	STATE_HV_ON:				BOOL;			(*Haute tension en marche*)
	STATE_HV:					BOOL;			(*Demande de mise en marche de la Haute Tension en cours*)
	STATE_SRC_ON:				BOOL;			(*Source en marche*)
	STATE_SRC:					BOOL;			(*Demande de mise en marche de la source en cours*)
	STATE_NOK:					BOOL;			(*Alimentation en défaut*)
	STATE_I_Fil:				REAL;			(*Mesure Courant filament (A)*)
	STATE_V_HV:					REAL;			(*Mesure de la tension (kV)*)
	STATE_I_EMISS:				REAL;			(*Mesure du courant d'émission (mA)*)
	STATE_COURANT:				REAL;			(* Courant appliqué en % *)
	STATE_READY:				BOOL;
END_VAR

VAR
END_VAR

HV.IdParent := MNEMO;
SRC.IdParent := MNEMO;
HV.IdXML := '16';
HV.TagXML := 1;
SRC.IdXML := '16';
SRC.TagXML := 2;
HV.MNEMO := 	CONCAT(MNEMO,'_HV');
SRC.MNEMO :=	CONCAT(MNEMO,'_SRC');

(*Défaut*)
HV.DEF_Off.IdXML				:=	'3';
HV.DEF_Off.TagXML				:=	3;
HV.DEF_On.IdXML				:=	'3';
HV.DEF_On.TagXML				:=	1;
HV.DEF_Off_Auto.IdXml			:=	'3';
HV.DEF_Off_Auto.TagXml			:=	10;
HV.DEF_On_imposs.IdXml		:=	'3';
HV.DEF_On_imposs.TagXml		:=	5;
HV.DEF_Off_imposs.IdXml		:=	'3';
HV.DEF_Off_imposs.TagXml		:=	8;

SRC.DEF_Off.IdXML				:=	'3';
SRC.DEF_Off.TagXML			:=	3;
SRC.DEF_On.IdXML				:=	'3';
SRC.DEF_On.TagXML			:=	1;
SRC.DEF_Off_Auto.IdXml			:=	'3';
SRC.DEF_Off_Auto.TagXml		:=	10;
SRC.DEF_On_imposs.IdXml		:=	'3';
SRC.DEF_On_imposs.TagXml		:=	5;
SRC.DEF_Off_imposs.IdXml		:=	'3';
SRC.DEF_Off_imposs.TagXml		:=	8;


HV(
	RESET:= RESET,
	MANUAL:= MANUAL,
	IN_ON:= NOT IN_HV_ON,
	CO_On:= CO_HV,
	EN_On_INT:=DOOR AND WATER AND VAC,
	EN_Off_INT:= TRUE,
	CONF_Type_Actuator:= 0,
	CONF_EN_On:= 0,
	CONF_DI_Off:= FALSE,
	CONF_DI_On:= TRUE,
	CONF_No_Safety_Auto:= FALSE,
	CONF_Tim_Valid_On:= T#2s,
	CONF_Tim_Valid_Off:= T#50ms,
	OUT_On=>OUT_HV,
	STATE_On=> STATE_HV_ON );
	
HV.DEF_Off.DELAY := T#10s;
HV.DEF_On.DELAY := T#10s;

STATE_HV := HV.OUT_On;

SRC(
	RESET:= RESET,
	MANUAL:= MANUAL,
	CO_On:=CO_SRC,
	IN_ON:= NOT IN_SRC_ON,
	EN_On_INT:=DOOR AND WATER  AND VAC AND (I_CR_OK OR (STATE_COURANT= 0)) AND STATE_HV_ON,
	EN_Off_INT:= TRUE,
	CONF_Type_Actuator:= 0,
	CONF_EN_On:= 0,
	CONF_DI_Off:= FALSE,
	CONF_DI_On:= TRUE,
	CONF_No_Safety_Auto:=FALSE ,
	CONF_Tim_Valid_On:= T#2s,
	CONF_Tim_Valid_Off:= T#50ms,
	OUT_On=>OUT_SRC,
	STATE_On=>STATE_SRC_ON );
	
SRC.DEF_Off.DELAY := T#10s;
SRC.DEF_On.DELAY := T#10s;

STATE_SRC := SRC.OUT_On;

AI_UHV(
	CONF_Max:= 10.0,
	CONF_Min:= 0.0,
	CONF_Bipolar:=FALSE,
	CONF_Range:= 1,
	INPUT:= IN_UHVQ ,
	Value=> STATE_V_HV );

AI_IEM(
	CONF_Max:= 1000,
	CONF_Min:= 0.0,
	CONF_Bipolar:=FALSE,
	CONF_Range:= 1,
	INPUT:= IN_IEMQ,
	Value=> STATE_I_EMISS );

AI_FIL(
	CONF_Max:= 100,
	CONF_Min:= 0.0,
	CONF_Bipolar:=FALSE ,
	CONF_Range:= 1,
	INPUT:= IN_FILQ ,
	Value=> STATE_I_Fil );

(*Gestion de la sortie analogique de courant d'emission*)
IF NOT STATE_SRC_ON OR RESET THEN
	AO_QIEM.Value := 0.0;
ELSIF MANUAL THEN
	AO_QIEM.Value := PRM_COURANT;
ELSE
	AO_QIEM.Value := I_COURANT;
END_IF;
STATE_COURANT:= AO_QIEM.Value;

AO_QIEM(
	CONF_Max:=100,  (*%*)
	CONF_Min:= 0,
	CONF_Bipolar:=FALSE ,
	CONF_Range:=1 ,
	OUTPUT=> OUT_QIEM );

(*Gestion de la sortie analogique haute tension*)
IF RESET THEN
	AO_QUHV.Value := 0.0;
ELSIF MANUAL THEN
	AO_QUHV.Value := PRM_TENSION;
ELSE
	AO_QUHV.Value := I_TENSION;
END_IF;

AO_QUHV(
	CONF_Max:=10,
	CONF_Min:= 0,
	CONF_Bipolar:=FALSE ,
	CONF_Range:=1 ,
	OUTPUT=> OUT_QUHV );

(*Gestion des interlock*)
OUT_ITLCK_VAC := DOOR AND VAC;
OUT_ITLCK_HVAC := DOOR AND VAC;
OUT_ITLCK_WAT := WATER;


STATE_NOK:= HV.STATE_Nok OR SRC.STATE_Nok;
STATE_READY:= WATER AND DOOR AND VAC AND I_CR_OK;

END_FUNCTION_BLOCK

// ---- POUs/FONCTION DE BASE/ANALOG_INPUT.TcPOU
FUNCTION_BLOCK ANALOG_INPUT
(* Fonction standard AC de mise à l'échelle *)

(****************historique des versions*****************************)

(* Version 1-0 - HG - VERSION INIITIALE*)

(*************************************************************************)
VAR_INPUT  PERSISTENT
	CONF_Max:	 			REAL;				(* ~ (OPC : 1 : available for OPC-clients) *)			(*valeur min*)
	CONF_Min: 				REAL:=0.0;			(* ~ (OPC : 1 : available for OPC-clients) *)			(*valeur max*)
	CONF_Bipolar:			BOOL:= FALSE;													(*option conversion en bipolaire (+/- 10V par ex) ou non (0-10V)*)
	CONF_Range:				REAL:=1;														(*Facteur de conversion par ex 0.5 pour une entrée ana 5V = pleine echelle*)
END_VAR

VAR_INPUT
 	INPUT:				 	INT;					(* ~ (OPC : 1 : available for OPC-clients) *)			(*entrée analogique*)
END_VAR

VAR_OUTPUT
	Value:					REAL;				(* ~ (OPC : 1 : available for OPC-clients) *)			(*value analogique convertie*)
END_VAR

IF CONF_Range = 0.0 THEN
	Value	:=	0;
	RETURN;
END_IF
IF CONF_Bipolar THEN
	Value	:=	(((INT_TO_REAL(INPUT) -32768.0)  * (CONF_Max-CONF_Min) / 65535.0 )  + CONF_Min) / CONF_Range;
ELSE
	Value	:=	((INT_TO_REAL(INPUT)   * (CONF_Max-CONF_Min) / 32767.0 )  + CONF_Min) / CONF_Range;
END_IF;

END_FUNCTION_BLOCK

// ---- POUs/FONCTION DE BASE/ANALOG_OUTPUT.TcPOU
FUNCTION_BLOCK ANALOG_OUTPUT
(* Fonction standard AC de mise à l'échelle *)

(****************historique des versions*****************************)

(* Version 1-0 - SP - VERSION INIITIALE*)

(*************************************************************************)
VAR_INPUT  PERSISTENT
	CONF_Max:	 			REAL;														(*valeur min*)
	CONF_Min: 				REAL:=0.0;													(*valeur max*)
	CONF_Bipolar:			BOOL:= FALSE;												(*option conversion en bipolaire (+/- 10V par ex) ou non (0-10V)*)
	CONF_Range:				REAL:=1;													(*Facteur de conversion par ex 0.5 pour une entrée ana 5V = pleine echelle*)
END_VAR

VAR_INPUT
 	Value:					REAL;				(* ~ (OPC : 1 : available for OPC-clients) *)		(*entrée analogique*)
END_VAR

VAR_OUTPUT
	OUTPUT:					INT ;				(* ~ (OPC : 1 : available for OPC-clients) *)		(*value analogique convertie*)
END_VAR

IF (CONF_Max-CONF_Min) = 0 THEN
	OUTPUT := 0;
	RETURN;
END_IF
IF CONF_Bipolar THEN
	OUTPUT := REAL_TO_INT((((Value - CONF_Min)*65536.0 / (CONF_Max-CONF_Min))+ 32767.0) * CONF_range);
ELSE
	OUTPUT := REAL_TO_INT(((Value - CONF_Min) * 32767.0 / (CONF_Max - CONF_Min)) * CONF_Range);
END_IF;

END_FUNCTION_BLOCK

// ---- POUs/Composant/EVAP/BLOCK_SOURCE_JOULE.TcPOU
FUNCTION_BLOCK BLOCK_SOURCE_JOULE
VAR_INPUT
	DOOR:						BOOL;		(*porte fermée*)
	VAC:						BOOL;		(*sécurité vide*)
	WATER:						BOOL;		(*refroidissement source ok*)
	MANUAL:					BOOL;		(*demande mode manuel*)
	I_CR_OK:					BOOL;		(*Positionnement creuset ok*)
	RESET:						BOOL;		(*reset*)

	AI_UEJ:						ANALOG_INPUT;
	AI_IEJ:						ANALOG_INPUT;

	IN_IEJQ			AT%I*:		INT;			(* Entrée analogique courant*)
	IN_UEJQ			AT%I*:		INT;			(* Entrée analogique tension*)

	EJ:							BLOCK_ACTUATOR2;		(*Source Effet Joule*)

	I_POWER:					REAL;		(*consigne de puissance appliquée en mode automatique*)
	PRM_POWER:				REAL;		(*Consigne de puissance appliquée en mode manuel*)
	CO_SRC:					BOOL;		(*Commande externe de marche de la source en automatique*)

END_VAR

VAR_INPUT PERSISTENT
	(*Entité*)
	IsComponent:		BOOL;			(*entité : composant*)
	IdXML:			STRING;			(*nom entité : identifiant pour recherche dans dico*)
	TagXML:			UINT;			(*nom entité : identifiant pour recherche dans dico*)
	IdParent:			STRING;			(*MNEMO de l'appelant*)
	MNEMO:			STRING;			(*MNEMO de l'entité*)
END_VAR

VAR_OUTPUT
	OUT_MEJ			AT%Q*:		BOOL;		(*Marche Effet joule*)

	AO_QEJ:				ANALOG_OUTPUT;		(*Sortie analogique consigne effet joule*)
	OUT_QEJ			AT%Q*:		INT;			(*Consigne effet joule*)

	STATE_UEJ:			REAL;			
	STATE_IEJ:			REAL;			
	
	
	STATE_EJ_ON:		BOOL;			(*Etat effet joule en marche*)

	STATE_POWER:		REAL;			(*Puissance appliquée en %*)

	STATE_NOK:			BOOL;			(*Alimentation en défaut*)
	STATE_READY:		BOOL;
END_VAR
VAR
END_VAR

EJ.IdParent := MNEMO;
EJ.IdXML := '16';
EJ.TagXML := 11;
EJ.MNEMO := 	CONCAT(MNEMO,'_EJ');

(*Défaut*)
EJ.DEF_Off_Auto.IdXml			:=	'3';
EJ.DEF_Off_Auto.TagXml		:=	10;
EJ.DEF_On_imposs.IdXml		:=	'3';
EJ.DEF_On_imposs.TagXml	:=	5;
EJ.DEF_Off_imposs.IdXml		:=	'3';
EJ.DEF_Off_imposs.TagXml	:=	8;


EJ(
	RESET:= RESET,
	MANUAL:= MANUAL,
	CO_On:=CO_SRC ,
	EN_On_INT:=DOOR AND WATER AND VAC AND (I_CR_OK OR (STATE_POWER = 0)),
	EN_Off_INT:= TRUE,
	CONF_No_Safety_Auto:=FALSE ,
	CONF_EN_On:= ,
	CONF_Tim_Valid_On:= T#5s,
	CONF_Tim_Valid_Off:= T#50ms,
	OUT_On=>,
	STATE_On=> ,
	STATE_Nok=> );

(*Demande marche Effet Joule*)
OUT_MEJ:= EJ.OUT_On;
STATE_EJ_ON:= OUT_MEJ;


(*Gestion de la sortie analogique*)
IF NOT STATE_EJ_ON OR RESET THEN
	AO_QEJ.Value := 0.0;
ELSIF MANUAL THEN
	AO_QEJ.Value := PRM_POWER;
ELSE
	AO_QEJ.Value := I_POWER;
END_IF;

AO_QEJ(
	CONF_Max:=100 ,	(*%*)
	CONF_Min:= 0,
	CONF_Bipolar:=FALSE ,
	CONF_Range:=1 );
OUT_QEJ:= AO_QEJ.OUTPUT;

STATE_POWER:= AO_QEJ.Value;

(*Retour Source en défaut*)
STATE_NOK:= EJ.STATE_Nok;
STATE_READY:= WATER AND DOOR AND VAC AND I_CR_OK;

(*Gestion de la sortie analogique source effet joule *)

AI_UEJ(
	CONF_Max:= 30.0,
	CONF_Min:= 0.0,
	CONF_Bipolar:=FALSE,
	CONF_Range:= 1,
	INPUT:= IN_UEJQ ,
	Value=> STATE_UEJ );

AI_IEJ(
	CONF_Max:= 500.0,
	CONF_Min:= 0.0,
	CONF_Bipolar:=FALSE,
	CONF_Range:= 1,
	INPUT:= IN_IEJQ ,
	Value=> STATE_IEJ );

END_FUNCTION_BLOCK

// ---- POUs/Composant/EVAP/BLOCK_TELEMARK_CHEETAH_SWEEP.TcPOU
FUNCTION_BLOCK BLOCK_TELEMARK_CHEETAH_SWEEP

(* Gestion d'un controleur de balayage telemark Digital Sweep 8 motifs*)

(****************historique des versions*****************************)

(* Version 1-0 - LDS - 01/09/26 - VERSION INIITIALE EVA900 n°1 - 5236 *)


(*************************************************************************)

VAR_INPUT
	MANUAL:					BOOL;		(*Mode de pilotage manuel *)
	RESET:					BOOL;		(*Condition de réinitialisation de la fonction *)
	DOOR:					BOOL;		(*Porte fermée*)
	
	I_SW_RUN:				BOOL;		(*Balayage en marche*)
	I_SW_RDY:				BOOL;		(*Balayage prêt*)
	
	PRM_NbBal:				USINT:=1;	(*Commande de position*)
	
	CO_Remote:				BOOL;		(*Demande d'activation du mode remote en automatique*)
	CO_Balayage:			BOOL;		(*Demande d'activation du balayage*)
END_VAR

VAR
	TIMER_Valid_On:			TON;
	TIMER_Valid_Off:		TOF;
	M_Remote:				BOOL;	(* Ordre de changement commande remote *)
	RCP_M_Remote:			BOOL;	(* Bit de reception de l'ordre de remote du module de balayage*)
	VAR_Remote:				BOOL;	(* Variable intermédiaire commande remote du module de balayage*)
	
	M_balayage:				BOOL;	(* Ordre de balayage en manuel*)
	RCP_M_Balayage:			BOOL;	(* Bit de reception de l'ordre de balayage du module de balayage*)
	VAR_Balayage:			BOOL;	(* Variable intermédiaire commande balayage du module de balayage*)
END_VAR

VAR_OUTPUT
	OUT_SWB1:			BOOL;		(*sélection du motif*)
	OUT_SWB2:			BOOL;		(*sélection du motif*)
	OUT_SWB3:			BOOL;		(*sélection du motif*)
	OUT_SWB4:			BOOL;		(*sélection du motif*)
	OUT_SWP_ON:			BOOL;		(*SWEEP ON/OFF*)
	OUT_RMT:			BOOL;		(*Remote*)
	STATE_NbBal:		USINT;
	STATE_BAL:			STRING;
	STATE_REM:			BOOL;		(*Module de balayage en mode Remote*)
	STATE_LOC:			BOOL;		(*Module de balayage en mode Local*)
	STATE_ON:			BOOL;		(*Module de balayage en marche*)
	STATE_OFF:			BOOL;		(*Module de balayage à l'arrêt*)
	STATE_RDY:			BOOL;		(*Module de balayage à prêt*)
	AUTOR_Remote_IHM:			BOOL;		(*indique que le changement mode remote est autorisé en mode manuel depuis l'IHM*)
	AUTOR_Remote_PLC:			BOOL;		(*indique que le changement more remote est autorisé en mode automatique depuis l'automate*)
	AUTOR_BALAYAGE_IHM:			BOOL;		(*indique que le changement mode remote est autorisé en mode manuel depuis l'IHM*)
	AUTOR_BALAYAGE_PLC:			BOOL;		(*indique que le changement more remote est autorisé en mode automatique depuis l'automate*)
END_VAR


VAR_INPUT PERSISTENT

	PRM_BAL: 		ARRAY[0..8] OF STRING;		(*nom du programme de balayage*)

	(*Entité*)
	IsComponent:	BOOL;			(*entité : composant*)
	IdXML:			STRING;			(*nom entité : identifiant pour recherche dans dico*)
	TagXML:			UINT;			(*nom entité : identifiant pour recherche dans dico*)
	IdParent:		STRING;			(*MNEMO de l'appelant*)
	MNEMO:			STRING;			(*MNEMO de l'entité*)
END_VAR

(* Gestion des ordres en mode manuel *)
RCP_M_Remote			:=	M_Remote;
RCP_M_Balayage			:=	M_Balayage;

(*affectation des bits d'état*)
STATE_REM			:=	OUT_RMT;
STATE_LOC			:=	NOT OUT_RMT;
STATE_OFF			:=	NOT I_SW_RUN;
STATE_RDY			:=	I_SW_RDY;

(*indicateur  STATE_ON*)

TIMER_Valid_On.IN	:=	I_SW_RUN;
TIMER_Valid_On(PT:=T#500ms);
TIMER_Valid_Off.IN	:=	I_SW_RUN;
TIMER_Valid_Off(PT:=T#200ms);
STATE_ON			:=	Timer_Valid_On.Q AND TIMER_Valid_Off.Q;

(*gestion des bits d'autorisation en mode manuel*)
AUTOR_Remote_IHM		:=	NOT RESET AND MANUAL;
AUTOR_Remote_PLC		:=	NOT RESET AND NOT MANUAL;
AUTOR_Balayage_IHM		:=	NOT RESET AND MANUAL;
AUTOR_Balayage_PLC		:=	NOT RESET AND NOT MANUAL;

(*Selection du mode de balayage*)
CASE PRM_NbBal OF
		8:
			OUT_SWB1 := FALSE;
			OUT_SWB2 := FALSE;
			OUT_SWB3 := FALSE;
			OUT_SWB4 := TRUE;
		7:
			OUT_SWB1 := TRUE;
			OUT_SWB2 := TRUE;
			OUT_SWB3 := TRUE;
			OUT_SWB4 := FALSE;
		6:
			OUT_SWB1 := FALSE;
			OUT_SWB2 := TRUE;
			OUT_SWB3 := TRUE;
			OUT_SWB4 := FALSE;
		5:
			OUT_SWB1 := TRUE;
			OUT_SWB2 := FALSE;
			OUT_SWB3 := TRUE;
			OUT_SWB4 := FALSE;
		4:
			OUT_SWB1 := FALSE;
			OUT_SWB2 := FALSE;
			OUT_SWB3 := TRUE;
			OUT_SWB4 := FALSE;
		3:
			OUT_SWB1 := TRUE;
			OUT_SWB2 := TRUE;
			OUT_SWB3 := FALSE;
			OUT_SWB4 := FALSE;
		2:
			OUT_SWB1 := FALSE;
			OUT_SWB2 := TRUE;
			OUT_SWB3 := FALSE;
			OUT_SWB4 := FALSE;
		1:
			OUT_SWB1 := TRUE;
			OUT_SWB2 := FALSE;
			OUT_SWB3 := FALSE;
			OUT_SWB4 := FALSE;
END_CASE
STATE_NbBal := PRM_NbBal;
IF STATE_NbBal > 0 THEN
	STATE_BAL:= PRM_BAL[STATE_NbBal];
ELSE
	STATE_BAL:= '';
END_IF

(*gestion SWP ON*)
IF	(CO_balayage AND AUTOR_BALAYAGE_PLC)
		 OR 	(RCP_M_Balayage AND NOT VAR_BALAYAGE AND AUTOR_BALAYAGE_IHM) THEN
			VAR_BALAYAGE 		:= 	TRUE;
ELSIF (NOT Co_balayage AND NOT RESET AND NOT MANUAL)
		OR 	(RCP_M_Balayage AND VAR_BALAYAGE AND AUTOR_BALAYAGE_IHM)
		OR 	RESET THEN
			VAR_BALAYAGE		:=	FALSE;
END_IF;
OUT_SWP_ON	:=	VAR_BALAYAGE;


(*gestion remote*)
IF	(CO_Remote AND AUTOR_Remote_PLC)
		 OR 	(RCP_M_Remote AND NOT VAR_Remote AND AUTOR_Remote_IHM) THEN
			VAR_Remote 		:= 	TRUE;
ELSIF (NOT CO_Remote AND NOT RESET AND NOT MANUAL)
		OR 	(RCP_M_Remote AND VAR_Remote AND AUTOR_Remote_IHM)
		OR 	RESET THEN
			VAR_Remote		:=	FALSE;
END_IF;
OUT_RMT	:=	VAR_Remote;

(* Reset des ordres*)
IF M_Remote	AND RCP_M_Remote THEN
	M_Remote			:=	FALSE;
END_IF

(* Reset des ordres*)
IF M_Balayage AND RCP_M_Balayage THEN
	M_Balayage		:=	FALSE;
END_IF

END_FUNCTION_BLOCK

// ---- POUs/Composant/EVAP/BLOCK_IND_CR_396_TELEMARK.TcPOU
FUNCTION_BLOCK BLOCK_IND_CR_396_TELEMARK

(* Pour utilisation d'un indexeur de creuset telemark 396/398 à 6 creusets max *)

(****************historique des versions*****************************)

(* Version 0 - 21/03/19 - GV - Affaire: 11385 - Block de base : BLOCK_IND_CR_379_TELEMARK *)

(*************************************************************************)

VAR_INPUT

	MANUAL:					BOOL;		(*Mode de pilotage manuel *)
	RESET:					BOOL;		(*Condition de réiinitialisation de la fonction *)

	CO_Change:				BOOL;		(*Demande de changement de creuset en automatique*)
	CO_Remote:				BOOL;
	I_FIL_ON:				BOOL;
	PRM_NCR:				USINT:=1;	(*Commande de position*)

	IN_POWER:				REAL;		(*Puissance appliquée au creuset*)

	IN_POS1:				BOOL;		(*position de l'indexeur*)
	IN_POS2:				BOOL;
	IN_POS3:				BOOL;
	IN_POS4:				BOOL;		(*position de l'indexeur*)
	IN_POS5:				BOOL;
	IN_POS6:				BOOL;
	IN_POS_OK:				BOOL;

	DEF_POSITIONNEMENT:	PRCDEF;	(*Défaut de positionnement*)
END_VAR

VAR
	VAR_Cpt_Temps:				ARRAY[0..8] OF BLOCK_CPT_TEMPS;		(*Compteur de fonctionnement pour chaque creuset*)
	VAR_Cpt_Puissance:			ARRAY[0..8] OF BLOCK_CPT_INTEG;		(*Compteur pour chaque creuset*)
	VAR_Cpt_Epaisseur:			ARRAY[0..8] OF BLOCK_CPT_INTEG;		(*Compteur d'épaisseur pour chaque creuset*)
	I:							USINT;									(*Variable d'itération*)

	M_Change:					BOOL;	(* Ordre de changement de creuset en manuel *)
	RCP_M_Change:				BOOL;	(* Bit de reception de l'ordre de Marche/Arrêt du module de balayage *)
	VAR_Change:					BOOL;	(* Variable intermédiaire de marche du module de balayage*)
	M_Remote: 					BOOL;
	RCP_M_Remote:				BOOL;
	VAR_Remote:					BOOL;
	
	TIMER_Valid_Pos_Creuset:		TON;	(*Attentede validation du positionnement du creuset*)
	FM_CO_remote:  				R_trig;
	FM_CO_Change:				r_trig;
	VAR_Mem_CO_remote:BOOL;
	VAR_Mem_CO_change:bool;
END_VAR

VAR_OUTPUT
	AUTOR_Change_IHM:			BOOL;		(*indique que le changement de creuset est autorisée en mode manuel depuis l'IHM*)
	AUTOR_Change_PLC:			BOOL;		(*indique que le changement de creuset est autorisée en mode automatique depuis l'automate*)
	AUTOR_Remote_IHM:			BOOL;		
	AUTOR_Remote_PLC:			BOOL;
	
	OUT_SEL1:					BOOL;		(*sélection  des creusets*)
	OUT_SEL2:					BOOL;
	OUT_SEL3:					BOOL;
	OUT_SEL4:					BOOL;		(*sélection  des creusets *)
	OUT_SEL5:					BOOL;
	OUT_SEL6:					BOOL;
	OUT_RMT:					BOOL;		(*force remote*)
	STATE_ROT:					BOOL;		(*Creuset en rotation*)
	STATE_NOK:					BOOL;		(*Positionnement nok*)
	STATE_POS_OK:				BOOL;		(*Positionnement ok*)
	STATE_POS:					USINT;
	STATE_MAT:					STRING;
	STATE_REM:					BOOL;		(*Remote OK*)
END_VAR

VAR_INPUT PERSISTENT
	CONF_NCR:		USINT;	(*Nombre de creuset disponible*)

	PRM_MAT: 		ARRAY[0..8] OF STRING;		(*nom de la matière associée au creuset*)

	(*Entité*)
	IsComponent:		BOOL;			(*entité : composant*)
	IdXML:			STRING;			(*nom entité : identifiant pour recherche dans dico*)
	TagXML:			UINT;			(*nom entité : identifiant pour recherche dans dico*)
	IdParent:			STRING;			(*MNEMO de l'appelant*)
	MNEMO:			STRING;			(*MNEMO de l'entité*)
END_VAR

(*Défaut*)
DEF_POSITIONNEMENT.IdXml			:=	'14';
DEF_POSITIONNEMENT.TagXml		:=	2;


(* Gestion des ordres en mode manuel *)
	RCP_M_Change			:=	M_Change;
	RCP_M_Remote			:=  M_remote;


	
(*gestion des bits d'autorisation en mode manuel*)
	AUTOR_Change_IHM		:=	NOT RESET AND NOT Var_Change AND NOT I_FIL_ON AND MANUAL;
	AUTOR_Change_PLC		:=	NOT RESET AND NOT I_FIL_ON AND NOT MANUAL;
	AUTOR_Remote_IHM		:=	NOT RESET AND MANUAL;
	AUTOR_Remote_PLC		:=	NOT RESET AND NOT MANUAL;	

(*gestion des variables intermédiare*)

(*Changement Creuset*)
	IF	(CO_change AND AUTOR_Change_PLC AND NOT var_change)								/////////
			 OR 	( RCP_M_Change AND AUTOR_Change_IHM) THEN
				Var_Change 		:= 	TRUE;
	ELSIF (VAR_Change AND STATE_POS_OK) THEN
				Var_Change		:=	FALSE;
	END_IF;
	
(*Remote*)	
IF (CO_remote AND AUTOR_Remote_PLC AND NOT var_remote) 									/////////
	OR (RCP_M_remote AND NOT var_remote AND AUTOR_Remote_IHM) THEN
		VAR_remote:=TRUE;
ELSIF (NOT CO_remote AND NOT reset AND NOT manual ) 
		OR (RCP_M_Remote AND VAR_Remote AND AUTOR_Remote_IHM)
		OR reset THEN
		VAR_Remote:=FALSE;
END_IF

IF PRM_NCR > CONF_NCR THEN
	PRM_NCR := CONF_NCR;
END_IF

IF VAR_Change THEN
	CASE PRM_NCR OF
			8:	OUT_SEL1 := FALSE;
				OUT_SEL2 := FALSE;
				OUT_SEL3 := FALSE;
				OUT_SEL4 := TRUE;
				OUT_SEL5 := FALSE;
				OUT_SEL6 := FALSE;
			7:
				OUT_SEL1 := TRUE;
				OUT_SEL2 := TRUE;
				OUT_SEL3 := TRUE;
				OUT_SEL4 := FALSE;
				OUT_SEL5 := FALSE;
				OUT_SEL6 := FALSE;
			6:
				OUT_SEL1 := FALSE;
				OUT_SEL2 := TRUE;
				OUT_SEL3 := TRUE;
				OUT_SEL4 := FALSE;
				OUT_SEL5 := FALSE;
				OUT_SEL6 := FALSE;
			5:
				OUT_SEL1 := TRUE;
				OUT_SEL2 := FALSE;
				OUT_SEL3 := TRUE;
				OUT_SEL4 := FALSE;
				OUT_SEL5 := FALSE;
				OUT_SEL6 := FALSE;
			4:
				OUT_SEL1 := FALSE;
				OUT_SEL2 := FALSE;
				OUT_SEL3 := TRUE;
				OUT_SEL4 := FALSE;
				OUT_SEL5 := FALSE;
				OUT_SEL6 := FALSE;
			3:
				OUT_SEL1 := TRUE;
				OUT_SEL2 := TRUE;
				OUT_SEL3 := FALSE;
				OUT_SEL4 := FALSE;
				OUT_SEL5 := FALSE;
				OUT_SEL6 := FALSE;
			2:
				OUT_SEL1 := FALSE;
				OUT_SEL2 := TRUE;
				OUT_SEL3 := FALSE;
				OUT_SEL4 := FALSE;
				OUT_SEL5 := FALSE;
				OUT_SEL6 := FALSE;
			1:
				OUT_SEL1 := TRUE;
				OUT_SEL2 := FALSE;
				OUT_SEL3 := FALSE;
				OUT_SEL4 := FALSE;
				OUT_SEL5 := FALSE;
				OUT_SEL6 := FALSE;
	END_CASE;
END_IF

(*affectation sotrie remote*)
OUT_RMT:=	 VAR_remote;

IF IN_POS1 AND NOT IN_POS2 AND NOT IN_POS3 AND NOT IN_POS4 AND NOT IN_POS5 AND NOT IN_POS6 THEN
		STATE_POS := 1;
ELSIF IN_POS2 AND NOT IN_POS1 AND NOT IN_POS3 AND NOT IN_POS4 AND NOT IN_POS5 AND NOT IN_POS6 THEN
		STATE_POS := 2;
ELSIF IN_POS1 AND IN_POS2 AND NOT IN_POS3 AND NOT IN_POS4 AND NOT IN_POS5 AND NOT IN_POS6 THEN
		STATE_POS := 3 ;
ELSIF IN_POS3 AND NOT IN_POS1 AND NOT IN_POS2 AND NOT IN_POS4 AND NOT IN_POS5 AND NOT IN_POS6 THEN
		STATE_POS := 4;
ELSIF IN_POS1 AND IN_POS3 AND NOT IN_POS2 AND NOT IN_POS4 AND NOT IN_POS5 AND NOT IN_POS6 THEN
		STATE_POS := 5;
ELSIF IN_POS2 AND IN_POS3 AND NOT IN_POS1 AND NOT IN_POS4 AND NOT IN_POS5 AND NOT IN_POS6 THEN
		STATE_POS := 6;
ELSIF IN_POS1 AND IN_POS2 AND IN_POS3 AND NOT IN_POS4 AND NOT IN_POS5 AND NOT IN_POS6 THEN
		STATE_POS := 7;
ELSIF IN_POS4 AND NOT IN_POS1 AND NOT IN_POS2 AND NOT IN_POS3 AND NOT IN_POS5 AND NOT IN_POS6 THEN
		STATE_POS := 8;
END_IF;



(*Attente de validation positionnement creuset*)
TIMER_Valid_Pos_Creuset.IN	:=	IN_POS_OK AND (PRM_NCR = STATE_POS);
TIMER_Valid_Pos_Creuset(PT:=T#500ms);
STATE_POS_OK	:= TIMER_Valid_Pos_Creuset.Q;

(*affectation des bits d'état*)
STATE_REM:=		OUT_RMT;
STATE_ROT:=	NOT IN_POS_OK;

DEF_POSITIONNEMENT.CONDITION :=  NOT IN_POS_OK;
DEF_POSITIONNEMENT.DELAY := T#180s;
DEF_POSITIONNEMENT();

(*gestion compteur d'utilisation*)
FOR I := 1 TO 8 BY 1 DO
	VAR_Cpt_Puissance[I].CONF_Coeff:=1;
	VAR_Cpt_Puissance[I].CONF_TimeUnit:=2;
	VAR_Cpt_Puissance[I].I_Value := IN_POWER;
	VAR_Cpt_Puissance[I].I_On := (STATE_POS = I);
	VAR_Cpt_Puissance[I]();

	VAR_Cpt_Temps[I].I_On := (STATE_POS = I) AND I_FIL_ON;		(*Compteur d'utilisation des creusets*)
	VAR_Cpt_Temps[I]();
END_FOR

STATE_NOK:= DEF_POSITIONNEMENT.DEF;

IF STATE_POS > 0 AND STATE_POS <= CONF_NCR THEN
	STATE_MAT:= PRM_MAT[STATE_POS];
ELSE
	STATE_MAT:= '';
END_IF

(* Reset des ordres*)
IF M_Change	AND RCP_M_Change THEN
	M_Change			:=	FALSE;
END_IF
IF M_Remote AND RCP_M_remote THEN
	M_remote := FALSE;
END_IF

END_FUNCTION_BLOCK

// ---- POUs/Fonction/FONCTIONS COMPTEUR/BLOCK_CPT_INTEG.TcPOU
FUNCTION_BLOCK BLOCK_CPT_INTEG
(* fonction permettant d'integrer une variable par rapport au temps*)
(* le comptage s'effectue lorsque l'entrée I_on est à true*)
(* on mesure les tick du processeur (1tick = 100ns) entre 2 appel du block = DeltaT*)
(* on ajoute au compteur la valeur mesurée en unité U sur I_value * DeltaT (en seconde) *)
(* le compteur VAR_CPT est exprimé en U*s ou U*min ou U*heure en fonction de la valeur du paramètres CONF_time_Unit *)
(* on peut convertir la valeur dans une unite (Wh en kWh par exemple) en fixant le paramètre CONF_coef (à 0.001 dans le cas de l'exémple)*)

(* Version 2.0 - SP - BA8 - 7326*)

VAR_INPUT
	I_On:						BOOL;			(*donne si la fonction appelante est dans l'état marche (true) ou arret (false) *)
	I_Value:					REAL;

END_VAR

VAR
	MEM_PREVIOUS_ON:			BOOL;		(*mémorise l'état antérieur*)
	VAR_Date_Off:				T_ULARGE_INTEGER;
	VAR_Date_On:				T_ULARGE_INTEGER;
	_GetCpuCounter:				FW_GetCpuCounter;

END_VAR

VAR_OUTPUT

END_VAR

VAR_INPUT PERSISTENT
	TagXML:				UINT;
	DISABLE:			BOOL;					(*indique que le compteur est desactivé*)
	CONF_Coeff:			REAL;					(*Coefficient de correction pour conversion des unités d'affichage*)
	CONF_TimeUnit:				USINT;			(*unité de temps pour le compteur
												0 = seconde
												1 = minute
												2 = heure
												*)
	CONF_UNIT:					STRING;
END_VAR

VAR_TEMP

	_TIM1:						T_ULARGE_INTEGER;
	_TIM2:						LREAL;
	VAR1:						UDINT;
	VAR2:						UDINT;

END_VAR
VAR PERSISTENT
	VAR_CPT:					LREAL;
	STATE_CPT:					REAL;
END_VAR

IF DISABLE THEN
	RETURN;
END_IF


(*sur le front descendant ou cycliquement, on met à jour la valeur de temps toutes les minutes*)
IF I_On THEN
	(*Lecture de l'horloge courant*)
	_GetCpuCounter(
						dwCpuCntLo=>	VAR1  ,
						dwCpuCntHi=>	VAR2
				 );

	VAR_Date_Off.dwLowPart := UDINT_TO_DWORD(VAR1);
	VAR_DATE_Off.dwHighPart := UDINT_TO_DWORD(VAR2);
	(*si la variable était à 1 au cycle précédent  alors on calcul la valeur*)
	IF MEM_PREVIOUS_ON THEN
		_TIM1 := UInt64Sub64(VAR_DATE_OFF,VAR_DATE_ON);
		_TIM2 := UINT64_TO_LREAL(_TIM1) / 10000000;
		IF CONF_TimeUnit = 0 THEN
			STATE_CPT := STATE_CPT + LREAL_TO_REAL(_TIM2 * REAL_TO_LREAL(I_VALUE)*REAL_TO_LREAL(CONF_Coeff));
		ELSIF CONF_TimeUnit = 1 THEN
			STATE_CPT:=  STATE_CPT + LREAL_TO_REAL(_TIM2 * REAL_TO_LREAL(I_VALUE)*REAL_TO_LREAL(CONF_Coeff) / REAL_TO_LREAL(60));
		ELSIF CONF_TimeUnit = 2 THEN
			STATE_CPT:=  STATE_CPT + LREAL_TO_REAL(_TIM2 * REAL_TO_LREAL(I_VALUE)*REAL_TO_LREAL(CONF_Coeff) / REAL_TO_LREAL(3600));
		END_IF
	END_IF

	VAR_Date_On := VAR_Date_Off;
	MEM_PREVIOUS_ON := TRUE;
ELSE
	MEM_PREVIOUS_ON:=FALSE;
END_IF;

END_FUNCTION_BLOCK

// ---- POUs/Programme/BLOCK_PRG_MOUVEMENT_PS.TcPOU
FUNCTION_BLOCK BLOCK_PRG_MOUVEMENT_PS
VAR_INPUT
	ROTATION_PS:					BLOCK_ROTATION_CONTINUE_ATV;
	PRM_Vitesse:					REAL;		(*Consigne de vitesse en procédé*)

	IN_SAFETY_OFF		AT%I*:		BOOL;		(*Permet de shunter les sécurité*)
	IN_CPS				AT%I*:		BOOL;		(*Capteur positionnement PS*)
	IN_JOG				AT%I*:		BOOL;		(*mouvement porte ouverte*)
END_VAR
VAR_INPUT PERSISTENT
(* Entité*)
	IsAssembly:				 	BOOL;			(*entité de type fonction*)
	TagXml:						UINT;
	IdXml: 						STRING;
	IdParent: 					STRING;			(*MNEMO du pére*)
	MNEMO:						STRING;			(*MNEMO de cette entité *)

(*Configuration pour visu - moteur ROTATION*)
	CONF_Positionnement:		BOOL;			(*Moteur utilisé pour du positionnement*)
	CONF_Rotation:				BOOL;			(*Moteur utilisé pour de la rotation continu*)
	CONF_Balayage:				BOOL;			(*Moteur utilisé pour du balayage*)

END_VAR

VAR_OUTPUT
	STATE_Ar:					BOOL;			(*I__STANDARD -indique que la fonction est à l'arrêt*)
	STATE_Pos_Ps_ok:			BOOL;			(*I__STD -- Indique que le positionnement du PS est OK*)
	STATE_Def_IProc:			BOOL;			(*I_STANDARD -indique la présence d'un défaut entrainant l'arrêt du procédé*)

END_VAR
VAR
	VAR_IN_Position:			BOOL;
END_VAR

(*paramètres de structure*)
IdXml								:= '5';
TagXml								:= 0;
IdParent							:=	MACHINE.MNEMO;
MNEMO								:=	CONCAT(IdParent,'_ATV320');

(*Configuration pour la visu*)
CONF_Positionnement					:=	FALSE;
CONF_Rotation						:=	TRUE;
CONF_Balayage						:=	FALSE;

ROTATION_PS.CONF_C1					:=	FALSE;
ROTATION_PS.CONF_C2					:=	FALSE;

ROTATION_PS.IN_POS_C1				:=	IN_CPS;
ROTATION_PS.IN_MVT					:=	IN_JOG;

ROTATION_PS.PS.PRM_Rapport		:=	98;
ROTATION_PS.PS.MNEMO			:=	'PS';
ROTATION_PS.PS.I_Valid_INPUT	:=	TRUE;

(*Configuration vitesse PS*)
ROTATION_PS.CONF_VMIN			:=	1;
ROTATION_PS.CONF_VMAX			:= 	20;
ROTATION_PS.CONF_V_Door_Open	:=	4;
ROTATION_PS.CONF_V_Pos			:=	3;

(*Configuration positionnement*)
ROTATION_PS.DEF_Position.DELAY		:=	T#2M;
ROTATION_PS.CONF_Pos_AvantSup		:=	FALSE;
ROTATION_PS.CONF_Pos_Capt			:=	1;
ROTATION_PS.CONF_Pos_MarcheArriere	:=	FALSE;
ROTATION_PS.CONF_Tim_AvantSup		:=	T#0MS;
ROTATION_PS.CONF_Tim_MarcheArriere	:=	T#0MS;


(*Gestion du mode de pilotage*)
IF MACHINE.RQ_Ctrl_Ihm AND NOT PRG_POMPAGE.RQ_PREP_VENTIL THEN
	ROTATION_PS.CTRL_PLC := FALSE;
ELSIF MACHINE.RQ_Ctrl_Plc OR PRG_POMPAGE.RQ_PREP_VENTIL THEN
	ROTATION_PS.CTRL_PLC := TRUE;
END_IF

ROTATION_PS.OP_ARRET.ON_PLC := INIT_MACHINE.RQ_STOP_MVTS
								OR EXECPROC.RQ_FM_EXEC_STEP[12]
								OR MACHINE.RQ_Prep_Prod
								OR MAIN.STEP_EFFLUVAGE.RQ_STOP_ROTATION_PS
								OR MAIN.STEP_TIMER.RQ_STOP_ROTATION_PS
								OR (MAIN.STEP_TIMER.RQ_ROTATION_PS AND (PRM_vitesse = 0))
								OR MAIN.STEP_EMPILEMENT.RQ_STOP_ROTATION_PS
								OR (MAIN.STEP_EMPILEMENT.RQ_ROTATION_PS AND (PRM_vitesse = 0));

ROTATION_PS.OP_Rotation.ON_PLC := 	EXECPROC.RQ_FM_EXEC_STEP[11]
									OR MAIN.STEP_EFFLUVAGE.RQ_ROTATION_PS
									OR (MAIN.STEP_TIMER.RQ_ROTATION_PS AND (PRM_vitesse <> 0))
									OR (MAIN.STEP_EMPILEMENT.RQ_ROTATION_PS AND (PRM_vitesse <> 0));

ROTATION_PS.OP_Rotation.ENABLE_EXT := MACHINE.STATE_Auto;

(*transmission consigne vitesse en procédé, sinon mise au mini et non nulle*)
IF (MAIN.STEP_TIMER.RQ_ROTATION_PS AND (PRM_vitesse <> 0)) OR MAIN.STEP_EMPILEMENT.OP_RUN.EC THEN
	ROTATION_PS.PRM_vitesse	:=	PRM_Vitesse;
END_IF

(*Moteur de rotation*)
ROTATION_PS(
	RESET:= MACHINE.STATE_Off,
	MANUAL:= MACHINE.STATE_Manu ,
	I_DOOR:=PRG_POMPAGE.DOOR OR IN_SAFETY_OFF ,
	STATE_NOK=> );


STATE_Def_IProc		:=		ROTATION_PS.OP_ARRET.DEF_AUTO_ON.DEF OR ROTATION_PS.OP_ARRET.DEF_ON_REJECTED.DEF
							OR ROTATION_PS.OP_Rotation.DEF_AUTO_ON.DEF OR ROTATION_PS.OP_Rotation.DEF_ON_REJECTED.DEF
							OR ROTATION_PS.OP_POSITION.DEF_AUTO_ON.DEF OR ROTATION_PS.OP_POSITION.DEF_ON_REJECTED.DEF
							OR ROTATION_PS.PS.DEF_Variateur.DEF OR ROTATION_PS.PS.DEF_off_auto.DEF
							OR ROTATION_PS.DEF_Rotation.DEF OR ROTATION_PS.DEF_Position.DEF
							OR ROTATION_PS.DEF_Capt_C1.DEF OR ROTATION_PS.DEF_Capt_C2.DEF;

STATE_AR 			:= 		((MACHINE.STATE_Auto OR MACHINE.STATE_Prod) AND ROTATION_PS.OP_ARRET.OK)
							OR (MACHINE.STATE_Manu AND (ROTATION_PS.PS.OUT_Velocity =0));

STATE_Pos_Ps_ok		:=		ROTATION_PS.OP_Rotation.OK;

END_FUNCTION_BLOCK

// ---- POUs/Fonction/FONCTIONS MVTS/BLOCK_ROTATION_CONTINUE_ATV.TcPOU
{attribute 'call_after_init'}
FUNCTION_BLOCK BLOCK_ROTATION_CONTINUE_ATV
(* Gestion d'un porte substrat en rotation continue sur variateur altivar*)

(****************historique des versions*****************************************)

(* Version 0 - JBL - VERSION INIITIALE - 7341*)
(* Version 1 - HG - Version pour moteur ATV Schneider EtherCAT*)
(* Version 2 - HG - Correction bug + ajout arrêt sur ouverture porte*)


VAR_INPUT
	RESET:					BOOL;		(* Condition de réinitialisation de la fonction *)
	MANUAL:					BOOL;		(* Ordre de commmande manuel de la fonction *)
	CTRL_PLC:				BOOL;		(* Mode de contrôle de la fonction - 0 = contrôle depuis l'IHM - 1=contrôle depuis l'automate*)
(*sécurité*)
	I_DOOR:					BOOL;		(* Entrée d'interlock porte fermée*)
(*Capteur position*)
	IN_POS_C1	AT %I*:		BOOL;		(* Capteur position pour déchargement*)
	IN_POS_C2	AT %I*:		BOOL;		(* Capteur position pour déchargement*)
	IN_MVT		AT %I*:		BOOL;		(* Entrée pour mouvement porte ouverte*)
(*Paramètres*)
	PRM_vitesse:			REAL;
	
(*composant*)
	PS:						BLOCK_MOTEUR_ATV_ANA;
(*Opérations*)
	OP_ROTATION:			BLOCK_OPERATION;	(*Opération rotation continue*)
	OP_POSITION:			BLOCK_OPERATION;	(*Opération positionnement sur capteur*)
	OP_ARRET:				BLOCK_OPERATION;	(*Opération arrêt mouvement*)
(*Défauts*)
	DEF_AUTOR_ROT_DOOR:		PRCDEF;		(* rotation non autorisée car porte ouverte *)
	DEF_AUTOR_POS_DOOR:		PRCDEF;		(* positionnement non autorisé car porte ouverte *)
	DEF_AUTOR_ROT_PS:		PRCDEF;		(* rotation non autorisée car variateur en défaut *)
	DEF_AUTOR_POS_PS:		PRCDEF;		(* positionnement non autorisé car variateur en défaut *)
	DEF_Position:			PRCDEF;		(* défaut de positionnement, capteur non rencontré*)
	DEF_Rotation:			PRCDEF;		(* défaut de rotation, capteur non rencontré*)
	DEF_Capt_C1:			PRCDEF;		(* défaut capteur C1 non fonctionnel - non rencontré*)
	DEF_Capt_C2:			PRCDEF;		(* défaut capteur C2 non fonctionnel - non rencontré*)
	
	CO_Modif:				BOOL;		(*Demande modification en ligne*)
	M_On:					BOOL;
END_VAR

VAR_OUTPUT
	STATE_Vitesse:			REAL;		(*Consigne vitesse appliquée *)
	STATE_Ready:			BOOL;		(*Moteur prêt*)
	STATE_Nok:				BOOL;		(*Moteur en défaut*)
	STATE_AR:				BOOL;		(*Pas de mouvement en cours*)
	STATE_EC:				BOOL;		(*Mouvement en cours*)	
	STATE_Position:			REAL;		(*Simulée depuis temps de rotation*)	
END_VAR

VAR_INPUT PERSISTENT
	CONF_VMAX:				REAL;		(*Consigne vitesse max*)
	CONF_VMIN:				REAL;		(*Consigne vitesse min*)
	CONF_V_Door_Open:		REAL;		(*Consigne vitesse porte ouverte*)
	CONF_V_Pos:				REAL:=1;	(*Consigne vitesse positionnement*)
	CONF_Tim_AvantSup:		TIME;		(*Consigne temps marche avant sup après front descendant capteur*)
	CONF_Tim_MarcheArriere:	TIME;		(*Consigne temps marche arrière pour centrer la clavette*)
	CONF_Pos_Capt:			USINT;		(*Option positionnement pour arrêt:
											0: sur présence capteur
											1: front montant capteur
											2: front descendant capteur*)
	CONF_Pos_AvantSup:		BOOL;		(*Option positionnement pour temps marche avant supplémentaire*)
	CONF_Pos_MarcheArriere:	BOOL;		(*Option positionnement pour marche arrière pour centrer la clavette*)	
	
	
	CONF_C1:				BOOL;		(*Conf présence capteur 1 positionnement*) 
	CONF_C2:				BOOL;		(*Conf présence capteur 2 positionnement*) 	
	
	(*Entité*)
	isAssembly:		BOOL;			(*entité : fonction*)
	IdXML:			STRING;			(*nom entité : identifiant pour recherche dans dico*)
	TagXML:			UINT;			(*nom entité : identifiant pour recherche dans dico*)
	IdParent:		STRING;			(*MNEMO de l'appelant*)
	MNEMO:			STRING;			(*MNEMO de l'entité*)
END_VAR

VAR
	VAR_Cons_Vitesse:		REAL;		(*Mémorisation consigne vitesse*)
	VAR_Door_Open:			BOOL;		(*Mouvement porte ouverte en automatique*)
	RCP_M_ON:				BOOL;
	VAR_On_Manu:			BOOL;
	FM_CO_Modif:			R_TRIG;
	FD_DOOR:				F_TRIG;
	FM_JOG:					R_TRIG;
	FM_IHM:					R_TRIG;
	FD_CAPT:				F_TRIG;
	FM_CAPT:				F_TRIG;
	TIMER_Tick:				TON;		(*Simulation position*)
	TIMER_AvantSup:			TON;
	TIMER_DemiTour:			TON;
END_VAR

IdXML	:= '5';
TagXML	:=	0;

OP_ROTATION.IdXML	:=	'6';
OP_ROTATION.TagXML	:=	2;

OP_POSITION.IdXML	:=	'6';
OP_POSITION.TagXML	:=	1;

OP_ARRET.IdXML		:=	'0';
OP_ARRET.TagXML		:=	2;

DEF_AUTOR_POS_DOOR.IdXML	:=	'5';
DEF_AUTOR_POS_DOOR.TagXML	:=	18;
DEF_AUTOR_ROT_DOOR.IdXML	:=	'5';
DEF_AUTOR_ROT_DOOR.TagXML	:=	18;
DEF_AUTOR_ROT_PS.IdXML		:=	'5';
DEF_AUTOR_ROT_PS.TagXML		:=	20;
DEF_AUTOR_POS_PS.IdXML		:=	'5';
DEF_AUTOR_POS_PS.TagXML		:=	20;

DEF_Position.IdXML	:=	'5';
DEF_Position.TagXML	:=	1;
DEF_Rotation.IdXML	:=	'5';
DEF_Rotation.TagXML	:=	4;
DEF_Capt_C1.IdXML	:=	'5';
DEF_Capt_C1.TagXML	:=	21;
DEF_Capt_C1.Groupe	:=	1;
DEF_Capt_C2.IdXML	:=	'5';
DEF_Capt_C2.TagXML	:=	22;
DEF_Capt_C2.Groupe	:=	1;

(*Opération arrêt mvt*)
ACT_STOP();
(*Opération marche mvt*)
ACT_START();
(*Opération positionnement*)
ACT_POS();
(*Fin de bloc*)
POST();

ACTION ACT_POS:
(*OPERATION MARCHE positionnement PS*)

OP_POSITION(
	CTRL_PLC:=CTRL_PLC,
	RESET:= RESET,
	MANUAL:= MANUAL ,
	ENABLE_INT:= PS.STATE_Ready,
	RESTART_ENABLE_IF_OK:=TRUE ,
	N_STEP_OP_OK:= 8,
	N_STEP_OP_NOK:=9 );

(*appel de l'action de préparation de l'opération*)
OP_POSITION.PRL();

(*GRAFCET*)
(* initialisation du grafcet*)
IF 		OP_POSITION.Etape = 0
		THEN
				OP_POSITION.Etape.0 := TRUE;
(*repositionnement sur étape 0*)
ELSIF 	MANUAL OR RESET OR OP_ARRET.ETAPE.1 OR OP_ROTATION.Etape.2 OR VAR_Door_Open
		THEN
				OP_POSITION.Etape := 0;
				OP_POSITION.Etape.0:=TRUE;
(*étape 0-1*)
ELSIF 	OP_POSITION.Etape.0 AND OP_POSITION.MARCHE_OP
		THEN
				OP_POSITION.Etape.1:=TRUE;
				OP_POSITION.Etape.0:=FALSE;
(*étape 1-9*)
ELSIF	OP_POSITION.Etape.1 AND NOT I_DOOR
		THEN
				OP_POSITION.Etape.9:=TRUE;
				OP_POSITION.Etape.1:=FALSE;
(*étape 9-0*)
ELSIF	OP_POSITION.Etape.9
		THEN
				OP_POSITION.Etape.0:=TRUE;
				OP_POSITION.Etape.9:=FALSE;
(*étape 1-10*)
ELSIF	OP_POSITION.Etape.1 AND PS.STATE_NOK
		THEN
				OP_POSITION.Etape.10:=TRUE;
				OP_POSITION.Etape.1:=FALSE;
(*étape 10-0*)
ELSIF	OP_POSITION.Etape.10
		THEN
				OP_POSITION.Etape.0:=TRUE;
				OP_POSITION.Etape.10:=FALSE;
(*étape 1-2*)
ELSIF	OP_POSITION.Etape.1 AND I_DOOR
		THEN
				OP_POSITION.Etape.2:=TRUE;
				OP_POSITION.Etape.1:=FALSE;
(*étape 2-3*)
ELSIF	OP_POSITION.Etape.2 AND OP_ARRET.Etape.0 AND OP_ROTATION.Etape.0
		THEN
				OP_POSITION.Etape.3:=TRUE;
				OP_POSITION.Etape.2:=FALSE;
(*étape 3-4*)
ELSIF	OP_POSITION.Etape.3 AND PS.STATE_ON THEN
				OP_POSITION.Etape.4:=TRUE;
				OP_POSITION.Etape.3:=FALSE;
(*étape 4-5*)
ELSIF	OP_POSITION.Etape.4 AND
		((FD_CAPT.Q AND conf_pos_capt = 2)
			OR (FM_CAPT.Q AND conf_pos_capt = 1)
			OR (((IN_POS_C1 AND CONF_C1) OR (IN_POS_C2 AND CONF_C2)) AND conf_pos_capt = 0)) THEN
				OP_POSITION.Etape.5:=TRUE;
				OP_POSITION.Etape.4:=FALSE;
(*étape 5-6*)
ELSIF	OP_POSITION.Etape.5 AND (TIMER_AvantSup.Q OR NOT CONF_Pos_AvantSup) THEN
				OP_POSITION.Etape.6:=TRUE;
				OP_POSITION.Etape.5:=FALSE;
(*étape 6-7*)
ELSIF	OP_POSITION.Etape.6 AND PS.STATE_OFF AND CONF_Pos_MarcheArriere THEN
				OP_POSITION.Etape.7:=TRUE;
				OP_POSITION.Etape.6:=FALSE;
(*étape 6-8*)
ELSIF	OP_POSITION.Etape.6 AND PS.STATE_OFF AND NOT CONF_Pos_MarcheArriere THEN
				OP_POSITION.Etape.8:=TRUE;
				OP_POSITION.Etape.6:=FALSE;
(*étape 7-8*)
ELSIF	OP_POSITION.Etape.7 AND TIMER_Demitour.Q AND PS.STATE_OFF THEN
				OP_POSITION.Etape.8:=TRUE;
				OP_POSITION.Etape.7:=FALSE;
(*étape 8-1*)
ELSIF	OP_POSITION.Etape.8 AND OP_POSITION.MARCHE_OP THEN
				OP_POSITION.Etape.1:=TRUE;
				OP_POSITION.Etape.8:=FALSE;
END_IF;
(*cloture du traitement de l'opération*)
OP_POSITION.POST();
END_ACTION

ACTION ACT_START:
(*OPERATION MARCHE rotation PS*)

OP_ROTATION(
	CTRL_PLC:=CTRL_PLC,
	RESET:= RESET,
	MANUAL:= MANUAL ,
	ENABLE_INT := TRUE,
	RESTART_ENABLE_IF_OK:=TRUE ,
	N_STEP_OP_OK:= 4,
	N_STEP_OP_NOK:=5 );

(*appel de l'action de préparation de l'opération*)
OP_ROTATION.PRL();

(*GRAFCET*)
(* initialisation du grafcet*)
IF 		OP_ROTATION.Etape = 0
		THEN
				OP_ROTATION.Etape.0 := TRUE;
(*repositionnement sur étape 0*)
ELSIF 	MANUAL OR RESET OR OP_ARRET.ETAPE.1 OR OP_POSITION.Etape.2
		THEN
				OP_ROTATION.Etape := 0;
				OP_ROTATION.Etape.0:=TRUE;
(*étape 0-1*)
ELSIF 	OP_ROTATION.Etape.0 AND OP_ROTATION.MARCHE_OP
		THEN
				OP_ROTATION.Etape.1:=TRUE;
				OP_ROTATION.Etape.0:=FALSE;
(*étape 1-5*)
ELSIF	OP_ROTATION.Etape.1 AND NOT I_DOOR
		THEN
				OP_ROTATION.Etape.5:=TRUE;
				OP_ROTATION.Etape.1:=FALSE;
(*étape 5-0*)
ELSIF	OP_ROTATION.Etape.5
		THEN
				OP_ROTATION.Etape.0:=TRUE;
				OP_ROTATION.Etape.5:=FALSE;
(*étape 1-6*)
ELSIF	OP_ROTATION.Etape.1 AND PS.STATE_NOK
		THEN
				OP_ROTATION.Etape.6:=TRUE;
				OP_ROTATION.Etape.1:=FALSE;
(*étape 6-0*)
ELSIF	OP_ROTATION.Etape.6
		THEN
				OP_ROTATION.Etape.0:=TRUE;
				OP_ROTATION.Etape.6:=FALSE;
(*étape 1-2*)
ELSIF	OP_ROTATION.Etape.1 AND I_DOOR
		THEN
				OP_ROTATION.Etape.2:=TRUE;
				OP_ROTATION.Etape.1:=FALSE;
(*étape 2-3*)
ELSIF	OP_ROTATION.Etape.2 AND OP_ARRET.Etape.0 AND OP_POSITION.Etape.0
		THEN
				OP_ROTATION.Etape.3:=TRUE;
				OP_ROTATION.Etape.2:=FALSE;
(*étape 3-4*)
ELSIF	OP_ROTATION.Etape.3  THEN
				OP_ROTATION.Etape.4:=TRUE;
				OP_ROTATION.Etape.3:=FALSE;
(*étape 4-3*)
ELSIF	OP_ROTATION.Etape.4 AND (OP_ROTATION.MARCHE_OP OR FM_CO_Modif.Q) AND PS.STATE_ON THEN
				OP_ROTATION.Etape.3:=TRUE;
				OP_ROTATION.Etape.4:=FALSE;
END_IF;
(*cloture du traitement de l'opération*)
OP_ROTATION.POST();
END_ACTION

ACTION ACT_STOP:
(*OPERATION arret rotation PS*)

OP_ARRET(
	CTRL_PLC:= CTRL_PLC,
	RESET:= RESET,
	MANUAL:= MANUAL ,
	ENABLE_INT:=TRUE,
	ON_AUTO_INT:= (PS.CO_On AND PS.STATE_NOK) OR (PS.DEF_Variateur.DEF AND PS.CO_On),
	RESTART_ENABLE_IF_OK:=TRUE ,
	N_STEP_OP_OK:= 3,
	N_STEP_OP_NOK:=0 );

(*appel de l'action de préparation de l'opération*)
OP_ARRET.PRL();

(*GRAFCET*)
(* initialisation du grafcet*)
IF 		OP_ARRET.Etape = 0
		THEN
				OP_ARRET.Etape.0 := TRUE;
(*repositionnement sur étape 0*)
ELSIF 	MANUAL OR RESET OR OP_ROTATION.ETAPE.2 OR OP_POSITION.Etape.2 OR VAR_Door_Open
	
		THEN
				OP_ARRET.Etape := 0;
				OP_ARRET.Etape.0:=TRUE;
(*étape 0-1*)
ELSIF 	OP_ARRET.Etape.0 AND (OP_ARRET.MARCHE_OP OR DEF_Position.DEF OR DEF_Rotation.DEF OR FD_DOOR.Q)
		THEN
				OP_ARRET.Etape.1:=TRUE;
				OP_ARRET.Etape.0:=FALSE;
(*étape 1-2*)
ELSIF 	OP_ARRET.Etape.1 AND OP_ROTATION.Etape.0 AND OP_POSITION.Etape.0
		THEN
				OP_ARRET.Etape.2:=TRUE;
				OP_ARRET.Etape.1:=FALSE;
(*étape 2-3*)
ELSIF 	OP_ARRET.Etape.2
		THEN
				OP_ARRET.Etape.3:=TRUE;
				OP_ARRET.Etape.2:=FALSE;
(*étape 3-1 : rebouclage sur nouvelle demande*)
ELSIF 	OP_ARRET.Etape.3
		AND OP_ARRET.MARCHE_OP
		THEN
				OP_ARRET.Etape.1:=TRUE;
				OP_ARRET.Etape.3:=FALSE;			
END_IF;

(*cloture du traitement de l'opération*)
OP_ARRET.POST();
END_ACTION

ACTION POST:
(*Gestion demandes*)
FM_CO_Modif(clk:=CO_modif);
RCP_M_On	:=	M_On;

(*front capteur*)
FD_CAPT(
	CLK := (IN_POS_C1 AND CONF_C1) OR (IN_POS_C2 AND CONF_C2),
	);
FM_CAPT(
	CLK := (IN_POS_C1 AND CONF_C1) OR (IN_POS_C2 AND CONF_C2),
	);

(*Vérification consignes*)
IF	PRM_Vitesse > CONF_VMAX THEN
	PRM_Vitesse	:=	CONF_VMAX;
END_IF;

IF PRM_Vitesse < CONF_VMIN THEN
	PRM_Vitesse := CONF_VMIN;
END_IF

(*Ouverture porte pour arrêt mouvement*)
FD_DOOR(CLK := I_DOOR);

(*Rotation porte ouverte*)
VAR_Door_Open	:=	IN_MVT AND NOT I_DOOR AND NOT RESET AND NOT CTRL_PLC;

(*Rotation en manuel*)
IF MANUAL AND RCP_M_ON AND I_DOOR AND NOT VAR_On_Manu THEN
	VAR_On_Manu	:=	TRUE;
ELSIF NOT MANUAL OR (RCP_M_On AND MANUAL AND VAR_On_Manu) OR NOT I_DOOR OR PS.STATE_NOK THEN
	VAR_On_Manu	:=	FALSE;
END_IF

(*Pilotage mouvement*)
PS.CO_On				:=	OP_ROTATION.Etape.3 OR OP_ROTATION.Etape.4 OR OP_POSITION.Etape.3 OR OP_POSITION.Etape.4 OR OP_POSITION.Etape.5
							OR (OP_POSITION.Etape.7 AND NOT TIMER_DemiTour.Q) OR VAR_Door_Open OR VAR_On_Manu;

(*Consigne vitesse*)
IF OP_ROTATION.Etape.3 OR (MANUAL AND VAR_On_Manu) THEN
	PS.PRM_Vitesse	:=	PRM_vitesse;
ELSIF OP_POSITION.Etape.3 OR OP_POSITION.Etape.4 OR OP_POSITION.Etape.5 THEN
	PS.PRM_Vitesse	:=	CONF_V_Pos;
ELSIF OP_POSITION.Etape.7 THEN
	PS.PRM_Vitesse	:=	-CONF_V_Pos;
ELSIF VAR_Door_Open THEN
	PS.PRM_Vitesse	:=	CONF_V_Door_Open;
ELSIF RESET OR NOT PS.CO_On THEN
	PS.PRM_Vitesse	:=	0.0;
END_IF

STATE_Vitesse	:=	PS.STATE_VIT;

PS(
	RESET:= RESET,
	CONF_VMIN:=CONF_VMIN,
	CONF_VMAX:=CONF_VMAX,
	);
	
(*TIMER*)
TIMER_DemiTour(
	IN	:=	OP_POSITION.Etape.7,
	PT	:=	CONF_Tim_MarcheArriere,
	);
	
TIMER_AvantSup(
	IN	:=	OP_POSITION.Etape.5,
	PT	:=	CONF_Tim_AvantSup,
	);
	
(*SIMULATION POSITION*)
TIMER_Tick();
TIMER_Tick.IN	:=	PS.STATE_ON;
TIMER_Tick.PT	:=	T#100MS;
IF TIMER_Tick.Q THEN
	STATE_Position	:=	STATE_Position + (STATE_Vitesse * 6 * 0.2); 	(*360/60, tick 0.5s*)
	IF STATE_Position > 360 THEN
		STATE_Position	:=	STATE_Position - 360;
	END_IF
	TIMER_Tick.IN	:=	FALSE;
END_IF

(*DEFAUTS*)
DEF_AUTOR_POS_DOOR.CONDITION	:=	OP_POSITION.Etape.9;
DEF_AUTOR_POS_DOOR();
DEF_AUTOR_ROT_DOOR.CONDITION	:=	OP_ROTATION.Etape.5;
DEF_AUTOR_ROT_DOOR();
DEF_AUTOR_POS_PS.CONDITION		:=	OP_POSITION.Etape.10;
DEF_AUTOR_POS_PS();
DEF_AUTOR_ROT_PS.CONDITION		:=	OP_ROTATION.Etape.6;
DEF_AUTOR_ROT_PS();

(*Temps de positionnement trop long*)
DEF_Position.CONDITION			:=	OP_POSITION.Etape.4;
DEF_Position();

(*Rotation non effective car aucun capteur rencontré*)
DEF_Rotation.CONDITION			:=	OP_ROTATION.Etape.4 AND (NOT IN_POS_C1 AND CONF_C1) OR (NOT IN_POS_C2 AND CONF_C2);
DEF_Rotation.DELAY				:=	T#2M;
DEF_Rotation();

(*défaut capteur C1 non opérationnel*)
IF NOT IN_POS_C1 AND PS.CO_On AND (PS.PRM_Vitesse>0) AND CONF_C1 THEN
	DEF_Capt_C1.CONDITION	:=	TRUE;
ELSIF IN_POS_C1 OR NOT CONF_C1 OR NOT PS.CO_On THEN
	DEF_Capt_C1.CONDITION	:=	FALSE;
END_IF
DEF_Capt_C1.DELAY	:=	T#2M;
DEF_Capt_C1();

(*défaut capteur C2 non opérationnel*)
IF NOT IN_POS_C2 AND PS.CO_On AND (PS.PRM_Vitesse>0) AND CONF_C2 THEN
	DEF_Capt_C2.CONDITION	:=	TRUE;
ELSIF IN_POS_C2 OR NOT CONF_C2 OR NOT PS.CO_On THEN
	DEF_Capt_C2.CONDITION	:=	FALSE;
END_IF
DEF_Capt_C2.DELAY	:=	T#2M;
DEF_Capt_C2();

(*ETATS*)
STATE_AR	:=	NOT PS.CO_On;
STATE_EC	:=	OP_POSITION.EC OR NOT OP_ROTATION.AR OR VAR_Door_Open;
STATE_Nok	:=	DEF_AUTOR_POS_DOOR.DEF OR DEF_AUTOR_ROT_DOOR.DEF
				OR DEF_AUTOR_POS_PS.DEF OR DEF_AUTOR_ROT_PS.DEF
				OR DEF_Position.DEF OR DEF_Rotation.DEF
				OR DEF_Capt_C1.DEF OR DEF_Capt_C2.DEF;
STATE_Ready	:=	PS.STATE_Ready;

(*reset des demandes*)
CO_Modif	:=	FALSE;
M_On		:=	FALSE;
END_ACTION

END_FUNCTION_BLOCK

// ---- POUs/Composant/MVTS/BLOCK_MOTEUR_ATV_ANA.TcPOU
FUNCTION_BLOCK BLOCK_MOTEUR_ATV_ANA

(****************historique des versions*****************************)
(* Version 0-0 - LDS - VERSION INIITIALE - basée sur BLOCK_MOTEUR_ATV - Affaire Original 5236*)

VAR_INPUT
	RESET			: BOOL;			(* Reinitialisation de la fonction *)
	I_Valid_INPUT	: BOOL;			(* Entrees exploitables (conserve pour compat interface) *)
	CO_On			: BOOL;			(* Marche moteur (depuis le grafcet) *)
	PRM_Vitesse		: REAL;			(* Consigne vitesse (unite procede) *)
	PRM_Rapport		: REAL;			(* Rapport cinematique - conserve pour compat (non utilise en analogique) *)

	VPS11M		AT %I* : BOOL;	(* Retour TOR "moteur en route" (relais R1 ATV12 -> VPS11M) *)

	DEF_off_auto	: PRCDEF;		(* Defaut d'arret automatique *)
	DEF_Variateur	: PRCDEF;		(* Defaut variateur *)
END_VAR

VAR_OUTPUT
	OUT_Marche		AT %Q* : BOOL;	(* -> LI1 (MPS11) commande marche rotation *)
	OUT_Velocity	AT %Q* : INT;	(* -> AI1 (QMPS11) consigne analogique 0..27648 (0-10 V) *)

	STATE_Ready		: BOOL;			(* Moteur pret *)
	STATE_OFF		: BOOL;			(* Moteur a l'arret *)
	STATE_EC		: BOOL;			(* Asservissement en cours (transition) *)
	STATE_ON		: BOOL;			(* Moteur en marche (retour confirme) *)
	STATE_NOK		: BOOL;			(* Moteur en defaut *)
	STATE_VIT		: REAL;			(* Vitesse appliquee *)
END_VAR

VAR_INPUT PERSISTENT
	CONF_VMAX		: REAL;			(* Consigne vitesse max = pleine echelle 10 V *)
	CONF_VMIN		: REAL;			(* Consigne vitesse min *)
	CONF_Deb_Retour	: TIME := T#300MS;	(* Anti-rebond du retour "moteur en route" *)
	CONF_Inv_Retour	: BOOL;			(* TRUE si le relais R1 est configure actif a 0 *)

	(* Entite *)
	IsComponent		: BOOL;
	IdXML			: STRING;
	TagXML			: UINT;
	IdParent		: STRING;
	MNEMO			: STRING;
END_VAR

VAR
	VAR_On		: BOOL;		(* marche moteur effective *)
	VAR_Marche	: BOOL;		(* retour normalise (polarite R1) *)
	TON_Route	: TON;		(* validation retour "en route" *)
	TON_Off		: TON;		(* validation "a l'arret" *)
END_VAR

(* ===== Parametre statique (identite dico, comme le bloc EtherCAT) ===== *)
IdXML				:= '5';
TagXML				:= 2;

DEF_off_auto.IdXML	:= '3';
DEF_off_auto.TagXML	:= 10;
DEF_Variateur.IdXML	:= '5';
DEF_Variateur.TagXML:= 4;

(* ===== Retour normalise (gestion polarite du relais R1) ===== *)
VAR_Marche := VPS11M XOR CONF_Inv_Retour;

(* ===== Verification des consignes (idem bloc EtherCAT) ===== *)
IF PRM_Vitesse > CONF_VMAX THEN
	PRM_Vitesse := CONF_VMAX;
END_IF
IF PRM_Vitesse < CONF_VMIN THEN
	PRM_Vitesse := CONF_VMIN;
END_IF

(* ===== Commande de marche -> LI1 ===== *)
VAR_On     := CO_On AND NOT RESET;
OUT_Marche := VAR_On;

(* ===== Consigne vitesse -> sortie analogique 0..32767 (0-10 V), unipolaire ===== *)
IF VAR_On AND (CONF_VMAX > 0.0) THEN
	OUT_Velocity := REAL_TO_INT(LIMIT(0.0, PRM_Vitesse / CONF_VMAX, 1.0) * 32767.0); (* PRM_Vitesse * PRM_Rapport ? *)
	STATE_VIT    := PRM_Vitesse;
ELSE
	OUT_Velocity := 0;
	STATE_VIT    := 0.0;
END_IF

(* ===== Anti-rebond du retour moteur ===== *)
TON_Route(IN := VAR_Marche,     PT := CONF_Deb_Retour);
TON_Off(  IN := NOT VAR_Marche, PT := CONF_Deb_Retour);

(* ===== Defaut variateur : marche commandee mais pas de retour, persistant CONF_Tempo_Def =====
   (sur ce cablage, R1 = "moteur en route", il n'existe pas de relais defaut dedie ;
    la temporisation est geree par le PRCDEF lui-meme via .DELAY) *)
DEF_Variateur.CONDITION	:= OUT_Marche AND NOT TON_Route.Q;
DEF_Variateur.DELAY		:= T#5S;
DEF_Variateur();

(* ===== Defaut d'arret automatique =====
   Pas de chaine de securite propre a ce terminal (geree en amont par le grafcet/porte).
   Neutralise ici ; le defaut significatif est DEF_Variateur. *)
DEF_off_auto.CONDITION := DEF_Variateur.DEF AND VAR_On;
DEF_off_auto.DELAY		:= T#0MS;
DEF_off_auto();

(* ===== Etats (memes semantiques que le bloc EtherCAT) ===== *)
STATE_ON	:= OUT_Marche AND TON_Route.Q AND NOT DEF_Variateur.DEF;
STATE_OFF	:= NOT OUT_Marche AND TON_Off.Q;
STATE_EC	:= NOT STATE_ON AND NOT STATE_OFF;
STATE_NOK	:= DEF_Variateur.DEF OR DEF_off_auto.DEF;
STATE_Ready	:= I_Valid_INPUT AND NOT RESET AND NOT STATE_NOK;

END_FUNCTION_BLOCK

// ---- POUs/Programme/BLOCK_PRG_POMPAGE.TcPOU
FUNCTION_BLOCK BLOCK_PRG_POMPAGE

(***********************************************************************************)
(* 		Programme pompage
		Pompage enceinte : cryo on-board + PPM 
		Vanne secondaire 2 positions
		Vanne primaire double avec une seule commande    


14035 - Pas de jauge Process M12 et sa vanne d'isolement VJ11	 *)
(***********************************************************************************)


VAR_INPUT
	POMPAGE:				BLOCK_POMP_1E_PCR_PPM_ASS_ETHERCAT_SINGER;
	//VJ11:					BLOCK_ACTUATOR;
	M11:					BLOCK_BCG450_ETHERCAT;
	//M12:					BLOCK_CDG_ETHERCAT;
	COM_CRYOS:				BLOCK_RS232_ONBOARD_V4;

	IN_FE11T	AT%I*:		BOOL;	(* ~ (OPC : 1 : available for OPC-clients) *)	(*Enceinte fermée - platine supérieure*)
	IN_FE12T	AT%I*:		BOOL;	(* ~ (OPC : 1 : available for OPC-clients) *)	(*Enceinte fermée - platine supérieure*)

	IN_ST11		AT%I*:		BOOL;	(* ~ (OPC : 1 : available for OPC-clients) *)	(*Pompe cryo en froid*)
	IN_ST12		AT%I*:		BOOL;	(* ~ (OPC : 1 : available for OPC-clients) *)	(*Pompe cryo en régénération*)

	IN_PP11M	AT%I*:		BOOL;	(* ~ (OPC : 1 : available for OPC-clients) *)	(*Pompe primaire en marche*)
	IN_PR11M	AT%I*:		BOOL;	(* ~ (OPC : 1 : available for OPC-clients) *)	(*Pompe roots enceinte en marche*)
	IN_PS11M	AT%I*:		BOOL;	(* ~ (OPC : 1 : available for OPC-clients) *)	(*Compresseur cryo en marche*)

	IN_VP11O	AT%I*:		BOOL;	(* ~ (OPC : 1 : available for OPC-clients) *)	(*Vanne pompage primaire rapide enceinte fermée*)
	IN_VP11F	AT%I*:		BOOL;	(* ~ (OPC : 1 : available for OPC-clients) *)	(*Vanne pompage primaire lente enceinte fermée*)
	
	IN_VS11F	AT%I*:		BOOL;	(* ~ (OPC : 1 : available for OPC-clients) *)	(*Vanne pompage secondaire enceinte fermée*)
	IN_VS11O	AT%I*:		BOOL;	(* ~ (OPC : 1 : available for OPC-clients) *)	(*Vanne secondaire enceinte ouverte*)
	IN_VS11Q	AT%I*:		INT;	(* ~ (OPC : 1 : available for OPC-clients) *)	(*Retour position vanne secondaire enceinte*)
	
//	IN_VJ11F	AT%I*:		BOOL;	(* ~ (OPC : 1 : available for OPC-clients) *)	(*Vanne isolement jauge fermée*)

	IN_M11Q		AT%I*:		REAL;	(* ~ (OPC : 1 : available for OPC-clients) *)	(*Pression enceinte *)
//	IN_M12Q		AT%I*:		REAL;	(* ~ (OPC : 1 : available for OPC-clients) *)	(*Pression procédé*)
	
	EV_DOOR: 				PRCDEF;	(* ~ (OPC : 1 : available for OPC-clients) *)	(*Evenement temps d'ouverture de la porte enceinte*)
END_VAR

VAR_INPUT PERSISTENT

(* Entité*)
	IsAssembly:				BOOL;			(*entité de type assemblage*)
	TagXml:					UINT;
	IdXml: 					STRING;
	IdParent: 				STRING;			(*MNEMO du pére*)
	MNEMO:					STRING;			(*MNEMO de cette entité *)

	CONF_WATER_ENC:			UINT:=0;		(*mot indiquant quelle ligne d'eau concerne le pompage enceinte .0 = ligne 1; .1 = ligne 2 ....*)
	CONF_N_Water_Line_PP11:	USINT;		(*index de la ligne d'eau affectée à la pompe PP11 - 0 = pas de ligne d'eau*)
	CONF_N_Water_Line_PR11:	USINT;		(*index de la ligne d'eau affectée à la pompe PP11 - 0 = pas de ligne d'eau*)
	CONF_N_Water_Line_PS11:	USINT;		(*index de la ligne d'eau affectée à la pompe PS11 - 0 = pas de ligne d'eau*)
	
	CONF_Tps_Pompage_Theorique: TIME;	(*Temps de pompage théorique pour calcul estimation temps procédé*)

	CONF_NO_FE12T:			BOOL;		(* option pas de capteur de fermeture enceinte FE11T*)
	CONF_NO_FE11T:			BOOL;		(* option pas de capteur de fermeture enceinte FE12T*)

	PRM_Min_Pumping_Time:	TIME;		(*I_STANDARD --- Temps de pompage min.*)
	PRM_Max_Pumping_Time:	TIME;		(*I_STANDARD ---- Temps de pompage max.*)
	PRM_Pr_Pumping_OK:		REAL;		(*I_STANDARD ---- Seuil de pression pour obtention étape de pompage OK*)

	PRM_Pr_Canon_OK:		REAL;		(*Seuil de pression pour autorisation allumage canon*)

END_VAR

VAR_OUTPUT
	OUT_PP11		AT%Q*:		BOOL;	(*Marche pompe primaire PP11*)
	OUT_PR11		AT%Q*:		BOOL;	(*Marche pompe roots*)
	OUT_PS11		AT %Q*:		BOOL;	(*Marche cryo enceinte*)

	OUT_VP111		AT%Q*:		BOOL;	(*Vanne primaire sortie 1*)
	OUT_VP112		AT%Q*:		BOOL;	(*Vanne primaire sortie 2*)

	OUT_OVS11		AT%Q*:		BOOL;	(*Ouverture vanne laminage*)
	OUT_FVS11		AT%Q*:		BOOL;	(*Fermeture vanne laminage*)
	OUT_LVS11		AT%Q*:		BOOL;	(*Laminage vanne laminage*)
	OUT_QVS11		AT%Q*:		INT;	(*Consigne position/pression vanne laminage*)
	
//	OUT_VJ11		AT%Q*:		BOOL;	(*Vanne d'isolement jauge capacitive*)

	OUT_VH11		AT%Q*:		BOOL;	(*Vanne de ventilation rapide enceinte*)

	OUT_VINT		AT%Q*:		BOOL;	(*Vanne de pompage interjoint*)

	OUT_DGZM11	AT%Q*:			BOOL;	(*Vanne de dégazage enceinte*)
	OUT_M11		AT%Q*:			BOOL;	(*Marche jauge secondaire enceinte*)
	
	OUT_VN2PP11	AT%Q*:		BOOL;	(*Vanne balayage pompe primaire pour évacuer l'humidité*)

	O_REF_ENC:				BOOL;	(*I_STANDARD --- Demande de refroidissement des élément lié à l'enceinte*)
	O_STEP_PUMPING_OK:		BOOL;	(*I_STANDARD --- information d'étape pompage secondaire ok*)

	VAC:					BOOL;	(*I_STANDARD --- Sécurité vide pour gaz / générateur / chauffage*)
	DOOR:					BOOL;	(*I_STANDARD --- Sécurité vide pour gaz / générateur / chauffage*)

	RQ_REF:					ARRAY[0..15] OF BOOL;	(*I_STANDARD -- demande de marche des lignes d'eau 1 à 8*)
	RQ_PREP_VENTIL:			BOOL;					(*I_STANDARD -- demande de réchauffement avant ventilation de l'enceinte*)

	STATE_Def_IProc:		BOOL;					(*I_STANDARD -indique la présence d'un défaut entrainant l'arrêt du procédé*)

END_VAR

VAR
	I:						USINT;		(*Variable d'iteration*)
	VAR_Mem_PS11_On:		BOOL;		(*mémorisation de l'état de PS11 en mode manuel*)
	VAR_debug_bool2:		BOOL;
	VAR_debug_bool3:		BOOL;
	TIMER_Reset_Memo_PSx1:	TON;		(*tempo lancée au passage en auto, on ne scrute plus la mémo des pompes, mais le prm_marche_groupe_x préalablement renseigné*)
	FM_EXEC_REGEN:			R_TRIG;
	
	TimeOpen    	: TIME;			(*Temps à l'ouverture de la porte*)
    TimeClose    	: TIME;			(*Temps à la fermeture de la porte*)
    TimeDifference	: TIME;			(*Temps d'ouverture de la chambre*)
	FM_DOOR			: R_TRIG;
	FD_DOOR			: F_TRIG;
	
	Tempo_on_Cryo: TON;
END_VAR

VAC			:=	M11.STATE_Seuil[3];
DOOR		:= 	(IN_FE11T OR CONF_NO_FE11T) AND (IN_FE12T OR CONF_NO_FE12T);

(*Calcule temps d'ouverture porte*)
FM_DOOR(CLK:= DOOR);
FD_DOOR(CLK:= DOOR);

IF FD_DOOR.Q THEN 
	TimeOpen:= TIME();
END_IF

IF FM_DOOR.Q THEN
	TimeClose:= TIME();
	TimeDifference:= TimeClose - TimeOpen;
END_IF

(*Evenement temps d'ouverture de la porte enceinte*)
EV_DOOR.IdXML 	:= '0';
EV_DOOR.TagXML 	:= 44;
EV_DOOR.Groupe 	:= 3;

EV_DOOR.VAL1 := DELETE(TIME_TO_STRING(TimeDifference), 2, 1);
EV_DOOR.CONDITION := FM_DOOR.Q;
EV_DOOR();

(*	Affectation des entrées 	 *)
POMPAGE.PP11.IN_On				:=	IN_PP11M;
POMPAGE.PR11.IN_On				:=	IN_PR11M;

POMPAGE.VS11.IN_ON 				:= 	IN_VS11O;
POMPAGE.VS11.IN_OFF				:=	IN_VS11F;
POMPAGE.VS11.IN_POSITION.INPUT 	:=	IN_VS11Q;
POMPAGE.VS11.I_PRESSION			:=	M11.STATE_Pression; 

IF NOT COM_CRYOS.STATE_NOK THEN            (* com OK  (STATE_NOK = DEF_Port_com.DEF) *)
    POMPAGE.PS11.IN_ON := IN_PS11M AND COM_CRYOS.STATE_Pompe;
ELSE                                       (* com perdue : retour degrade *)
    POMPAGE.PS11.IN_ON := IN_PS11M;
END_IF
POMPAGE.PS11.IN_ST11			:=	IN_ST11;
POMPAGE.PS11.IN_ST12			:=	IN_ST12;



//VJ11.IN_OFF						:=	IN_VJ11F;

POMPAGE.VP11.IN_OFF				:=	IN_VP11F;
POMPAGE.VP11.IN_ON				:=	IN_VP11O;

M11.IN_Pression					:=	IN_M11Q;
//M12.IN_Pression					:=	IN_M12Q;

(* Parametre statique *)
(*General*)
IdXML									:=	'2';
TagXML									:=	0;

CONF_NO_FE11T							:=	FALSE;
CONF_NO_FE12T							:=	TRUE;
CONF_WATER_ENC							:=	2#00000000;	

(*PP11*)
CONF_N_Water_Line_PP11				:=	5;
POMPAGE.PP11.CONF_Tim_Valid_Off 	:= 	T#100MS;
POMPAGE.PP11.CONF_Tim_Valid_On		:=	T#10s;
POMPAGE.PP11.DEF_On.DELAY			:=	T#10s;
POMPAGE.PP11.DEF_Off.DELAY			:=	T#5s;
POMPAGE.PP11.MNEMO					:=	'PP11';
POMPAGE.PRM_Tim_Arret_PP11			:=	T#30m;

(*PR11*)
CONF_N_Water_Line_PR11				:=	0;
POMPAGE.PR11.CONF_Tim_Valid_Off 	:= 	T#10S;
POMPAGE.PR11.CONF_Tim_Valid_On		:=	T#10S;
POMPAGE.PR11.DEF_On.DELAY			:=	T#15S;
POMPAGE.PR11.DEF_Off.DELAY			:=	T#15S;
POMPAGE.PR11.MNEMO					:=	'PR11';

(*PS11*)
CONF_N_Water_Line_PS11				:=	0;
POMPAGE.PS11.MNEMO					:=	'PS11';

(*VP11*)
POMPAGE.VP11.CONF_EN_On				:=	0;
POMPAGE.VP11.CONF_Tim_Valid_Off		:=	T#1S;
POMPAGE.VP11.CONF_Tim_Valid_On		:=	T#5S;
POMPAGE.VP11.DEF_Off.DELAY			:=	T#10S;
POMPAGE.VP11.DEF_On.DELAY			:=	T#10S;
POMPAGE.VP11.DEF_Lam.DELAY			:=	T#10S;
POMPAGE.VP11.MNEMO					:=	'VP11';
POMPAGE.VP11.CONF_DI_On				:=	TRUE;
POMPAGE.VP11.CONF_DI_Lam			:=	FALSE;
POMPAGE.VP11.CONF_DI_Off			:=	TRUE;
	
(*VS11*)
POMPAGE.VS11.CONF_Tim_Valid_Off		:=	T#1S;
POMPAGE.VS11.CONF_Tim_Valid_On		:=	T#1S;
POMPAGE.VS11.CONF_EN_On				:=	0;
POMPAGE.VS11.DEF_Position.DELAY		:=	T#20S;
POMPAGE.VS11.DEF_Off.DELAY			:=	T#10S;
POMPAGE.VS11.DEF_On.DELAY			:=	T#10S;
POMPAGE.VS11.MNEMO					:=	'VS11';
POMPAGE.VS11.CONF_Tim_WPos			:=	T#2S;		(*Temps de validation du positionnement ok*)
POMPAGE.VS11.CONF_WPos				:=	3.0;			(*Précision d'obtention de la position 3%*)
POMPAGE.VS11.CONF_Pr_Max_SP			:=	0.0665;

(*VH11*)
POMPAGE.VH11.CONF_DI_Off			:=	FALSE;
POMPAGE.VH11.CONF_DI_On				:=	FALSE;
POMPAGE.VH11.CONF_EN_On				:=	0;
POMPAGE.VH11.CONF_Tim_Valid_Off		:=	T#500ms;
POMPAGE.VH11.CONF_Tim_Valid_On		:=	T#500ms;
POMPAGE.VH11.CONF_Type_Actuator		:=	0;
POMPAGE.VH11.CONF_No_Safety_Auto	:=	FALSE;
POMPAGE.VH11.DEF_Off.DELAY			:=	T#10s;
POMPAGE.VH11.DEF_On.DELAY			:=	T#10s;
POMPAGE.VH11.MNEMO					:=	'VH11';

(*VINT*)
POMPAGE.VINT.CONF_DI_Off			:=	FALSE;
POMPAGE.VINT.CONF_DI_On				:=	FALSE;
POMPAGE.VINT.CONF_EN_On				:=	0;
POMPAGE.VINT.CONF_Tim_Valid_Off		:=	T#500ms;
POMPAGE.VINT.CONF_Tim_Valid_On		:=	T#500ms;
POMPAGE.VINT.CONF_Type_Actuator		:=	0;
POMPAGE.VINT.CONF_No_Safety_Auto	:=	FALSE;
POMPAGE.VINT.DEF_Off.DELAY			:=	T#10s;
POMPAGE.VINT.DEF_On.DELAY			:=	T#10s;
POMPAGE.VINT.MNEMO					:=	'VPINT';

(*VBAL*)
POMPAGE.VN2PP11.CONF_DI_Off				:=	FALSE;
POMPAGE.VN2PP11.CONF_DI_On				:=	FALSE;
POMPAGE.VN2PP11.CONF_EN_On				:=	0;
POMPAGE.VN2PP11.CONF_Tim_Valid_Off		:=	T#10S;
POMPAGE.VN2PP11.CONF_Tim_Valid_On		:=	T#500MS;
POMPAGE.VN2PP11.CONF_Type_Actuator		:=	0;
POMPAGE.VN2PP11.CONF_No_Safety_Auto		:=	FALSE;
POMPAGE.VN2PP11.DEF_Off.DELAY			:=	T#10S;
POMPAGE.VN2PP11.DEF_On.DELAY			:=	T#10S;
POMPAGE.VN2PP11.MNEMO					:=	'VN2PP11';

(*M11*)
M11.MNEMO								:=	'M11';

M11.PRM_Type_seuil[1]					:=	TRUE;			(* Seuil 1 = Pression > pression atm*)
M11.PRM_Delais[1]						:=	T#10s;
M11.PRM_Type_seuil[2]					:=	FALSE;			(* Seuil 2 = Pression <= Seuil détection grosse fuite*)
M11.PRM_Delais[2]						:=	T#500ms;
M11.PRM_Delais[3]						:=	T#10s;			(* Seuil 3 = Pression <= Pression de basculement en pompage secondaire*)
M11.PRM_Type_seuil[3]					:=	FALSE;
M11.PRM_Delais[4]						:=	T#500ms;		(* Seuil 4 = Pression >= Pression max. en pompage secondaire.*)
M11.PRM_Type_seuil[4]					:=	TRUE;
M11.PRM_Delais[5]						:=	T#2s;			(* Seuil 5 = Pression <= Pression max. pour autorisation transfert sous vide*)
M11.PRM_Type_seuil[5]					:=	FALSE;
M11.PRM_Delais[6]						:=	T#2S;			(* Seuil 6 = Pression <= Pression de basculement en pompage rapide*) (*utilisé pour interjoint*)
M11.PRM_Type_seuil[6]					:=	FALSE;
M11.PRM_Delais[7]						:=	T#200ms;		(* Seuil 7 = Pression <= Consigne pression étape de pompage *)
M11.PRM_Type_seuil[7]					:=	FALSE;
M11.PRM_Seuil[8] 						:= 	1E-0;
M11.PRM_Delais[8]						:=	T#2s;			(* Seuil 8 = Pression <= Pression max. sécurité générateur / gaz / chauffage*)
M11.PRM_Type_seuil[8]					:=	FALSE;
M11.PRM_Delais[9]						:=	T#2s;			(* Seuil 9 = Pression >= Pression de bascuelement en ventilation rapide*) (*Non utilisé*)
M11.PRM_Type_seuil[9]					:=	TRUE;
M11.PRM_Delais[10]						:=	T#2s;			(* Seuil 10 = Pression < Pression de mise en marche de la circulation d'eau froide dans l'enceinte*)
M11.PRM_Type_seuil[10]					:=	FALSE;
M11.PRM_Delais[11]						:=	T#2s;			(* Seuil 11 = Pression <= Pression test RP*)
M11.PRM_Type_seuil[11]					:=	FALSE;
M11.PRM_Delais[12]						:=	T#500ms;		(* Seuil 12 = Pression <= Seuil de pompage avant effluvage*)
M11.PRM_Type_seuil[12]					:=	FALSE;
M11.PRM_Delais[13]						:=	T#2s;
M11.PRM_Type_seuil[13]					:=  FALSE;			(* Seuil 13= Pression <= Pression de vide pour autorisation allumage canon*)
M11.PRM_Delais[14]						:=	T#2s;
M11.PRM_Type_seuil[14]					:=  FALSE;			(* Seuil 14= Pression <= Pression de vide pour autorisation allumage effluvage*)
M11.PRM_Delais[15]						:=	T#2S;
M11.PRM_Type_seuil[15]					:=	FALSE;			(* Seuil 15= Pression <= Pression basse pour autorisation allumage effluvage*)		


M11.CONF_Unit							:=	0 ;				(* mbar*)
M11.CONF_degas_auto						:= 	TRUE;
M11.CONF_Tim_Degas						:=	T#20S;
M11.PRM_Tim_Restart						:=	T#10S;
M11.PRM_Tim_Stop						:=	T#15s;
(*CoE*)
M11.CONF_NetId							:=	'172.18.237.251.2.1';
M11.CONF_SlaveAddr						:=	1029;

(*M12*)
(*M12.MNEMO								:=	'M12';
M12.CONF_Unit							:=	0 ;			(*mbar*)

(*VJ11*)
VJ11.MNEMO								:=	'VJ11';
VJ11.IdXML								:=	'2';
VJ11.TagXML								:=	4;
VJ11.DEF_On.IdXML						:=	'3';
VJ11.DEF_On.TagXML						:=	2;
VJ11.DEF_Off.IdXML						:=	'3';
VJ11.DEF_Off.TagXML						:=	4;
VJ11.DEF_Sensor.IdXML					:=	'3';
VJ11.DEF_Sensor.TagXML					:=	13;
VJ11.DEF_On_Imposs.IdXML				:=	'3';
VJ11.DEF_On_Imposs.TagXML				:=	6;
VJ11.DEF_Off_Imposs.IdXML				:=	'3';
VJ11.DEF_Off_Imposs.TagXML				:=	9;
VJ11.DEF_Off_auto.IdXML					:=	'3';
VJ11.DEF_Off_auto.TagXML				:=	11;

VJ11.DEF_Off.DELAY 						:= 	T#10s;
VJ11.DEF_On.DELAY 						:= 	T#10s;
VJ11.CONF_Type_Actuator					:=	0;
VJ11.CONF_EN_On							:=	0;
VJ11.CONF_DI_Off						:=	FALSE;
VJ11.CONF_DI_On							:= 	FALSE;
VJ11.CONF_No_Safety_Auto				:=	FALSE;
VJ11.CONF_Tim_Valid_On					:=	T#100ms;
VJ11.CONF_Tim_Valid_Off					:= 	T#100ms;*)

(*COM CRYOS*)
COM_CRYOS.MNEMO						:=	'COM_CRYOS';
COM_CRYOS.IdParent					:=	MNEMO;

(*mode de controle des fonctions*)
IF (MACHINE.RQ_Ctrl_Ihm OR MACHINE.STATE_Manu)
	AND NOT PRG_GAZ.REGULATION_GAZ_L1.RQ_Ctrl_Pompage
	AND NOT PRG_GAZ.REGULATION_GAZ_L2.RQ_Ctrl_Pompage THEN
	POMPAGE.CTRL_PLC := FALSE;
ELSIF (MACHINE.RQ_Ctrl_Plc AND NOT MACHINE.STATE_Manu)
		OR PRG_GAZ.REGULATION_GAZ_L1.RQ_Ctrl_Pompage
		OR PRG_GAZ.REGULATION_GAZ_L2.RQ_Ctrl_Pompage THEN
	POMPAGE.CTRL_PLC := TRUE;
END_IF


POMPAGE.OP_Marche_Pompes.ON_PLC  := INIT_MACHINE.RQ_START_PUMP
										OR EXECPROC.RQ_FM_EXEC_STEP[3];

POMPAGE.OP_Pompage_Sec.ON_PLC 	:= 	INIT_MACHINE.RQ_START_PUMPING
										OR EXECPROC.RQ_FM_EXEC_STEP[1]
										OR MAIN.STEP_EMPILEMENT.RQ_MARCHE_POMPAGE_SEC
										OR MAIN.STEP_EFFLUVAGE.RQ_POMPAGE_SEC
										OR PRG_GAZ.REGULATION_GAZ_L1.RQ_Pompage_Sec
										OR PRG_GAZ.REGULATION_GAZ_L2.RQ_Pompage_Sec;

POMPAGE.OP_Pompage_Prim.ON_PLC 	:=	MAIN.STEP_EFFLUVAGE.RQ_POMPAGE_PRIM;

POMPAGE.OP_Pompage_Proc.ON_PLC	:=	MAIN.STEP_EMPILEMENT.RQ_MARCHE_POMPAGE_PROC;

IF PRG_GAZ.REGULATION_GAZ_L1.RQ_Pompage_Proc THEN
	POMPAGE.VS11.PRM_Mode			:=	0;	(*asservissement en position*)
	POMPAGE.VS11.PRM_Position			:=	PRG_GAZ.REGULATION_GAZ_L1.PRM_Pos_Vanne;
	POMPAGE.OP_Pompage_Proc.ON_PLC :=	TRUE;
END_IF

IF PRG_GAZ.REGULATION_GAZ_L2.RQ_Pompage_Proc THEN
	POMPAGE.VS11.PRM_Mode			:=	0;	(*asservissement en position*)
	POMPAGE.VS11.PRM_Position			:=	PRG_GAZ.REGULATION_GAZ_L2.PRM_Pos_Vanne;
	POMPAGE.OP_Pompage_Proc.ON_PLC :=	TRUE;
END_IF

POMPAGE.OP_Arret_Pompes.ON_PLC := EXECPROC.RQ_FM_EXEC_STEP[4];
PRG_POMPAGE.POMPAGE.OP_Regen.ON_PLC  := EXECPROC.RQ_FM_EXEC_STEP[5];
PRG_POMPAGE.POMPAGE.OP_Regen_Part.ON_PLC := EXECPROC.RQ_FM_EXEC_STEP[19];
PRG_POMPAGE.POMPAGE.OP_Ventilation.ON_PLC := EXECPROC.RQ_FM_EXEC_STEP[6];
PRG_POMPAGE.POMPAGE.OP_Isolement.ON_PLC := EXECPROC.RQ_FM_EXEC_STEP[2] OR MAIN.STEP_EFFLUVAGE.RQ_ISOLEMENT;
PRG_POMPAGE.POMPAGE.OP_Test_RP.ON_PLC := EXECPROC.RQ_FM_EXEC_STEP[14];

(*Paramètre dynamique*)
(*PP11*)
POMPAGE.PP11.WATER					:=	PRG_SERVITUDES.WATER[CONF_N_Water_Line_PP11] AND NOT PRG_SERVITUDES.DEF_Groupe.DEF;
POMPAGE.PP11.EN_Off_EXT				:= 	TRUE;
POMPAGE.PP11.EN_On_EXT				:= 	TRUE;
(*PR11*)
POMPAGE.PR11.WATER					:=	PRG_SERVITUDES.WATER[CONF_N_Water_Line_PR11];
POMPAGE.PR11.EN_Off_EXT				:= 	TRUE;
POMPAGE.PR11.EN_On_EXT				:= 	TRUE;
(*PS11*)
POMPAGE.PS11.WATER					:=	PRG_SERVITUDES.WATER[CONF_N_Water_Line_PS11] AND NOT PRG_SERVITUDES.DEF_Groupe.DEF;
POMPAGE.PS11.EN_Off_EXT				:= 	TRUE;
POMPAGE.PS11.EN_On_EXT				:= 	TRUE;
(*VS11*)
POMPAGE.VS11.EN_Off_EXT				:=	TRUE;
POMPAGE.VS11.EN_On_EXT				:=	TRUE;
(*VP11*)
POMPAGE.VP11.EN_Off_EXT				:=	TRUE;
POMPAGE.VP11.EN_On_EXT				:=	TRUE;
(*VH11*)
POMPAGE.VH11.EN_Off_EXT				:=	TRUE;
POMPAGE.VH11.EN_On_EXT				:=	(*VJ11.STATE_Off AND*) PRG_EFFLUVAGE.STATE_Ar AND PRG_GAZ.STATE_Ar AND PRG_EVAP.STATE_Ar;


(*paramétrage déclenchement automatique opérations*)
POMPAGE.OP_Arret_Pompes.ON_AUTO_EXT	:= 	PRG_SERVITUDES.DEF_Groupe.DEF;

(*paramétrage opérations pompage*)
POMPAGE.OP_Ventilation.ENABLE_EXT		:=	PRG_EFFLUVAGE.STATE_Ar AND PRG_GAZ.STATE_Ar AND PRG_EVAP.STATE_Ar AND M11.STATE_Ok;
POMPAGE.OP_Isolement.ENABLE_EXT			:=	PRG_EFFLUVAGE.STATE_Ar AND PRG_GAZ.STATE_Ar AND PRG_EVAP.STATE_Ar ;
POMPAGE.OP_Arret_Pompes.ENABLE_EXT		:=	TRUE ;
POMPAGE.OP_Marche_Pompes.ENABLE_EXT		:=	TRUE;
POMPAGE.OP_Pompage_Prim.ENABLE_EXT		:=	TRUE ;
POMPAGE.OP_Pompage_Sec.ENABLE_EXT		:=	TRUE;
POMPAGE.OP_Pompage_Proc.ENABLE_EXT		:=	TRUE;
POMPAGE.OP_Purge.ENABLE_EXT				:=	TRUE;
POMPAGE.OP_Regen.ENABLE_EXT				:=	PRG_EFFLUVAGE.STATE_AR AND PRG_GAZ.STATE_Ar AND PRG_EVAP.STATE_AR;
POMPAGE.OP_Test_RP.ENABLE_EXT			:=	PRG_EFFLUVAGE.STATE_Ar AND PRG_GAZ.STATE_Ar AND PRG_EVAP.STATE_Ar AND M11.STATE_Ok;


(*Fonction pompage*)
POMPAGE.CONF_Pompage_interjoint		:= TRUE;
POMPAGE.CONF_VINT					:= TRUE;




(**************************************************************************************)
(*	                             Fonction pompage enceinte 					   *)
(**************************************************************************************)

(*DEBUGECO*)
IF VAR_Mem_ECO THEN
	IF EXECPROC.RQ_FM_EXEC_STEP[1] THEN
		DEBUG_BOOL1	:=	TRUE;
		IF POMPAGE.OP_Pompage_Sec.AUTOR_PLC	THEN
			DEBUG_BOOL2	:=	TRUE;
		ELSIF NOT POMPAGE.PS11.STATE_Regen THEN
			DEBUG_BOOL3	:=	TRUE;
		END_IF
	END_IF
	IF EXECPROC.RQ_EXEC_STEP[1] THEN
		DEBUG_BOOL4	:=	TRUE;
	END_IF
	IF EXECPROC.RQ_FM_EXEC_STEP[3] THEN
		DEBUG_BOOL5	:=	TRUE;
		IF POMPAGE.OP_Marche_Pompes.AUTOR_PLC	THEN
			DEBUG_BOOL6	:=	TRUE;
		END_IF
	END_IF
	IF EXECPROC.RQ_EXEC_STEP[3] THEN
		DEBUG_BOOL7	:=	TRUE;
	END_IF
END_IF

POMPAGE(
	RESET:=					MACHINE.STATE_Off ,
	MANUAL:= 				MACHINE.STATE_Manu,
	I_Prep_Ventil_Ok:= 		(NOT CONF_WATER_ENC.0 OR PRG_SERVITUDES.STATE_AR[1]) AND
							(NOT CONF_WATER_ENC.1 OR PRG_SERVITUDES.STATE_AR[2]) AND
							(NOT CONF_WATER_ENC.2 OR PRG_SERVITUDES.STATE_AR[3]) AND
							(NOT CONF_WATER_ENC.3 OR PRG_SERVITUDES.STATE_AR[4]) AND
							(NOT CONF_WATER_ENC.4 OR PRG_SERVITUDES.STATE_AR[5]) AND
							(NOT CONF_WATER_ENC.5 OR PRG_SERVITUDES.STATE_AR[6]) AND
							(NOT CONF_WATER_ENC.6 OR PRG_SERVITUDES.STATE_AR[7]) AND
							(NOT CONF_WATER_ENC.7 OR PRG_SERVITUDES.STATE_AR[8]),
	I_Fin_Ventil:= 			FALSE,
	I_Ref_Ok:=				NOT PRG_SERVITUDES.DEF_Groupe.DEF,
	I_Stop_Mesure_OK:= 		M11.O_Pret_Pour_Rah (*AND VJ11.STATE_Off*),
	I_Cond_Bal_PP11_Ext:=	PRG_EVAP.STATE_AR,
	IN_Pressure_RP:=		M11.STATE_Pression,
	IN_FE11T	:=			IN_FE11T OR CONF_NO_FE11T,
	IN_FE12T	:= 			IN_FE12T OR CONF_NO_FE12T,
	TH_Vide_Primaire:=		M11.STATE_Seuil[3] ,
	TH_Grosse_Fuite:= 		M11.STATE_Seuil[2],
	TH_Atm:= 				M11.STATE_Seuil[1],
	TH_RP_Enc:=				NOT M11.STATE_Seuil[4],
	TH_Test_RP:=			M11.STATE_Seuil[11],
	PRM_Tim_SurVentil_E:= ,	(*Affecté depuis IHM*)
	PRM_Tim_Purge:= ,		(*Affecté depuis IHM*)
	PRM_Pr_Atm:= ,			(*Affecté depuis IHM*)
	PRM_Pr_PPrim:= ,		(*Affecté depuis IHM*)
	PRM_Pr_RP_PPrim:= ,		(*Affecté depuis IHM*)
	PRM_Pr_TGF:= ,			(*Affecté depuis IHM*)
	PRM_N_Purge:= ,			(*Affecté depuis IHM*)
	PRM_Pr_test:=,			(*Affecté depuis IHM*)
	IN_Temp_Etage1 :=		COM_CRYOS.STATE_Temperature[0],
	 );


(*************************************************************************************)
(*                                   Jauge mesure pression enceinte M11                             *)
(*************************************************************************************)

(* Seuil 1 = Pression > pression atm*)
(* Seuil 2 = Pression <= Seuil détection grosse fuite*)
(* Seuil 3 = Pression <= Pression de basculement en pompage secondaire*)
(* Seuil 4 = Pression <= Pression max. en pompage secondaire.*)
(* Seuil 5 = Pression <= Pression MAX Sécurité transfert*) (*Non utilisé*)
(* Seuil 6 = Pression <= Pression de basculement en prévidage rapide*) (*Non utilisé*)
(* Seuil 7 = Pression <= Consigne pression étape de pompage *)
(* Seuil 8 = Pression <= Pression MAX. Sécurité générateur / gaz / chauffage*)
(* Seuil 9 = Pression > Pression de basculement en ventilation rapide*) (*Non utilisé*)
(* Seuil 10 = Pression < Pression de mise en marche de la circulation d'eau froide dans l'enceinte*)
(* Seuil 11 = Pression <= Pression test de remontée de pression*)
(* Seuil 12 = Pression <= Pression avant effluvage*)
(* Seuil 13= Pression <= Pression de vide pour autorisation allumage canon*)
(* Seuil 14= Pression <= Pression de vide pour autorisation allumage effluvage*)
(* Seuil 15= Pression => Pression basse pour autorisation allumage effluvage*)


(* Paramètre dynamique*)
M11.PRM_Seuil[1] :=			POMPAGE.PRM_Pr_Atm;
M11.PRM_Seuil[2] := 		POMPAGE.PRM_Pr_TGF;
M11.PRM_Seuil[3] := 		POMPAGE.PRM_Pr_PPrim;
M11.PRM_Seuil[4] :=			POMPAGE.PRM_Pr_RP_PPrim;
M11.PRM_Seuil[6] :=			100; 		
M11.PRM_Seuil[7]:=			PRM_Pr_Pumping_OK;
M11.PRM_Seuil[10] := 		PRG_SERVITUDES.PRM_Pr_REF_ENC;
M11.PRM_Seuil[11]:=			POMPAGE.PRM_Pr_test;
M11.PRM_Seuil[12]:=			MAIN.STEP_EFFLUVAGE.PRM_PR_EFFLUVAGE;
M11.PRM_Seuil[13]:=			PRM_Pr_Canon_Ok;
M11.PRM_Seuil[14]:=			1;
M11.PRM_Seuil[15]:=			5.0E-2;

M11(
	RESET:=					MACHINE.STATE_Off,
	MANUAL:= 				MACHINE.STATE_Manu,
	CO_Stop:= 				FALSE,
	CO_inhibe_Seuil:=		FALSE ,
	I_Stop_Rah:=			POMPAGE.RQ_Stop_Mesure_Enc ,
	I_VHxx:= 				POMPAGE.VH11.STATE_On,
	EN_Dgz_EXT:=			POMPAGE.OP_Pompage_sec.OK OR M11.MANUAL ,
	EN_Off_EXT:=			TRUE,
);


(***************************************************************************************************)
(*                   GESTION  DE LA VANNE D'ISOLEMENT JAUGE M12				      *)
(***************************************************************************************************)
(*VJ11(
	I_PARAM_SYSTEM_OK:=	PARAM_SYSTEM_OK,
	RESET:= 				MACHINE.STATE_Off,
	MANUAL:= 				MACHINE.STATE_Manu,
	CO_On:= 				M11.STATE_Seuil[3]  AND POMPAGE.OP_Ventilation.AR,
	EN_On_INT:= 			TRUE,
	EN_Off_INT:= 			TRUE,
	EN_On_EXT:= 			M11.STATE_Seuil[3]  AND POMPAGE.VH11.STATE_Off,
	EN_Off_EXT:= 			TRUE
	);*)

(***************************************************************************)
(*                              JAUGE CAPACITIVE M12                                        *)
(***************************************************************************)
(*M12(
	RESET:=				MACHINE.STATE_Off,
	MANUAL:= 			MACHINE.STATE_Manu,
	CO_inhibe_Seuil:=	FALSE ,
	);*)

(*************************************************************************************)
(*                        Communication pompes cryos				                    *)
(*************************************************************************************)
COM_CRYOS.CO_Regen			:=	POMPAGE.PS11.OUT_Regen;
COM_CRYOS.CO_Etat			:=	POMPAGE.PS11.OUT_On ;
COM_CRYOS.CO_states_regen 	:=  POMPAGE.PS11.STATE_Regen;
COM_CRYOS(
	RESET:= 				MACHINE.STATE_Off,
	OFF:= 					FALSE,
);


(* INFORMATION EN SORTIE DU PROGRAMME*)
O_REF_ENC		:=		M11.STATE_Seuil[10] AND POMPAGE.OP_Ventilation.AR;

(*Affectation des sorties*)
(*Vanne VP11.1 & VP11.2 même commande OUT_VP11*)
OUT_VP111		:= 		POMPAGE.VP11.OUT_V11;
OUT_VP112		:=		POMPAGE.VP11.OUT_V12;

OUT_OVS11		:=      POMPAGE.VS11.OUT_On;
OUT_FVS11		:=      POMPAGE.VS11.OUT_Off;
OUT_LVS11		:=      POMPAGE.VS11.OUT_Mode;
OUT_QVS11		:=      POMPAGE.VS11.OUT_SetPoint.OUTPUT;

OUT_VH11		:=		POMPAGE.VH11.OUT_On;
OUT_VINT		:=		POMPAGE.VINT.OUT_On;

OUT_PP11		:=		POMPAGE.PP11.OUT_On;
OUT_PR11		:=		POMPAGE.PR11.OUT_On;
OUT_PS11		:=		POMPAGE.PS11.OUT_On;

OUT_VN2PP11		:=		POMPAGE.VN2PP11.OUT_On;

(*OUT_VJ11		:=		VJ11.OUT_On;*)
(*
OUT_DGZM11	:=		M11.OUT_DGZ;
OUT_M11		:=		M11.OUT_M1;
*)
(*Gestion des demandes de refroidissements*)
FOR i:= 1 TO 8 DO
	RQ_REF[I]	:=	(POMPAGE.PP11.RQ_Cool  AND (I=CONF_N_Water_Line_PP11))
					OR (POMPAGE.PR11.RQ_Cool AND (I=CONF_N_Water_Line_PR11))
					OR (POMPAGE.PS11.RQ_Cool AND (I=CONF_N_Water_Line_PS11));
END_FOR
RQ_PREP_VENTIL	:=	POMPAGE.RQ_Prep_Ventil_Enc;

O_STEP_PUMPING_OK	:=	POMPAGE.OP_Pompage_Sec.OK AND M11.STATE_Seuil[7];


(*Défaut entrainant l'interruption du procédé*)
STATE_Def_IProc		:=	POMPAGE.OP_Arret_Pompes.DEF_AUTO_ON.DEF OR POMPAGE.OP_Isolement.DEF_AUTO_ON.DEF
						OR POMPAGE.OP_Pompage_Prim.DEF_ON_REJECTED.DEF OR POMPAGE.OP_Pompage_Sec.DEF_ON_REJECTED.DEF
						OR POMPAGE.OP_Pompage_Proc.DEF_ON_REJECTED.DEF OR POMPAGE.OP_Purge.DEF_ON_REJECTED.DEF
						OR POMPAGE.OP_Regen.DEF_ON_REJECTED.DEF
						OR POMPAGE.VS11.DEF_Surv_Pression.DEF OR POMPAGE.VS11.DEF_Pression.DEF OR POMPAGE.VS11.DEF_Position.DEF;

END_FUNCTION_BLOCK

// ---- POUs/Fonction/FONCTIONS POMPAGE/BLOCK_POMP_1E_PCR_PPM_ASS_ETHERCAT_SINGER.TcPOU
FUNCTION_BLOCK BLOCK_POMP_1E_PCR_PPM_ASS_ETHERCAT_SINGER

(* Historique des versions*)
(* VERSION 1.0 - 05/2015 - GV - affaire 9070*)
(* VERSION 2.0 - 10/2022 - GV - ajout gestion roots *)
(* VERSION 3.0 - 11/2023 - HG - ajout balayage pompe primaire en alternance avec interjoint (specif SINGER pour bcp d'humidité)
								ajout évènement résultat test de remontée de pression pour inscription dans le journal*)


(* BLOCK GESTION POMPAGE CRYO ON BOARD ENCEINTE *)
(*	Gestion pompage enceinte sans sas constitué de :
	Pompe primaire pour prévidage, regen cryo et pompage interjoint
	Pompe cryogénique on-board CTI pour le pompage secondaire
	Vanne de pompage primaire enceinte
	Vanne de remise à atmosphère enceinte
	Vanne de pompage inter-joint (optionnelle)
	Vanne secondaire asservie, pilote en ana
	Vanne de balayage pompe primaire
*)

VAR_INPUT
(*information générale*)
	RESET:					BOOL;
	MANUAL:					BOOL;
	CTRL_PLC:				BOOL;
	I_Prep_Ventil_Ok:		BOOL;		(*information externe indiquant que l'enceinte est prête à être ventilée par ex. circulation d'eau à l'arrêt
										ou polycold arreté ou basculement en eau chaude ok ...*)
	I_Fin_Ventil:			BOOL;		(*information externe de fin de ventilation de l'enceinte  *)
	I_Stop_Mesure_OK:		BOOL;		(*information externe indiquant que les jauges ont été stoppées prélablement à la ventilation de l'enceinte*)
	IN_Pressure_RP:			REAL;		(*interfaçage avec M11.state_pression du PRG correspondant*)
	I_Ref_OK:				BOOL;		(*information externe indiquant que le refroidissement est ok pour démarrer les pompes*)
	I_Cond_Bal_PP11_Ext:	BOOL;		(*information externe condition balayage pompe primaire - pas de chauffage/puissance/evap*)
	
(*Gestion régen partielle*)
	IN_Temp_Etage1:			REAL;
	PRM_Temp_Post_Purge:	REAL;
	PRM_Tim_Post_Purge:		TIME;

(*Paramètres et commandes du test de remontée de pression*)
	PRM_Pr_test:			REAL;		(*Pression initiale de test de remontée*)
	PRM_Tim_test:			TIME;		(*Durée d'attente en test*)
	CO_Stop_Test_RP:		BOOL;		(*Demande arrêt test remontée de pression*)

(*sécurité*)
	IN_FE11T:				BOOL;		(*indicateur enceinte fermée - capteur 1*)
	IN_FE12T:				BOOL;		(*indicateur enceinte fermée - capteur 2*)
	IN_VT11F:				BOOL;		(*clapet SAS enceinte fermé*)

(*seuil de vide*)
	TH_Vide_Primaire:		BOOL;		(*Pression enceinte <= Seuil de fin de pompage primaire*)
	TH_Grosse_Fuite:		BOOL;		(*Pression enceinte <= Seuil de detection de grosse fuite enceinte*)
	TH_Atm:					BOOL;		(*pression enceinte >= Seuil pression atm. de fin de ventilation*)
	TH_RP_Enc:				BOOL;		(*pression enceinte <= Pression max. dans l'enceinte*)
	TH_Test_RP:				BOOL;		(*Pression <= Seuil de pression de test*)
	TH_Ouv_VINT:			BOOL;		(*Pression enceinte <= seuil ouverture VINT*)

(*composant de la fonction*)
	VP11:					BLOCK_VVAT_3P;									(*vanne de pompage primaire enceinte *)
	VH11:					BLOCK_ACTUATOR;									(*vanne de ventilation de l'enceinte*)
	PP11:					BLOCK_PPM;										(*Pompe primaire enceinte*)
	PR11:					BLOCK_PPM;										(*Pompe roots enceinte*)
	PS11:					BLOCK_PCR_CTI_OB;								(*Pompe cryogénique on board  enceinte*)
	VS11:					BLOCK_VVAT_650_NO;								(*Vanne secondaire asservie pompage enceinte*)
	VINT:					BLOCK_ACTUATOR;									(*Vanne de pompage dans les interjoints*)
	VN2PP11:				BLOCK_ACTUATOR;									(*Vanne de balayage pompe primaire*)

(*défaut*)
	DEF_PPrim:				PRCDEF;										(*défaut temps de pompage primaire dans l'enceinte*)
	DEF_Vent:				PRCDEF;										(*défaut temps de ventilation enceinte*)
	DEF_RP_enc:				PRCDEF;	 									(*défaut perte seuil de pompage primaire en pompage secondaire*)
	DEF_TGF:				PRCDEF;										(*défaut détection trés grosse fuite*)
	EV_Test_RP:				PRCDEF;										(*évènement affichage résultate test RP*)

(*opération*)
	OP_Marche_Pompes:			BLOCK_OPERATION;								(*opération marche pompe*)
	OP_Arret_Pompes:			BLOCK_OPERATION;								(*opération arrêt pompe*)
	OP_Isolement:				BLOCK_OPERATION;								(*opération stand-by*)
	OP_Ventilation:				BLOCK_OPERATION;								(*opération ventilation*)
	OP_Pompage_Sec:				BLOCK_OPERATION;								(*opération pompage secondaire*)
	OP_Pompage_Prim:			BLOCK_OPERATION;								(*opération pompage primaire*)
	OP_Pompage_Proc:			BLOCK_OPERATION;								(*opération pompage en procédé*)
	OP_Purge:					BLOCK_OPERATION;								(*opération purge*)
	OP_Regen:					BLOCK_OPERATION;								(*opération régénération pompe cryogénique*)
	OP_Regen_Part:				BLOCK_OPERATION;								(*opération de régénération partielle pompe cryogénique*)
	OP_Test_RP:					BLOCK_OPERATION;								(*opération test RP*)
	G7_Bal_Int:					BLOCK_G7;										(*gestion balayage pompe primaire et pompage interjoint*)
	
END_VAR

VAR_INPUT PERSISTENT
(*paramètre*)
	PRM_Tim_SurVentil_E:		TIME;	(*durée du temps de surventilation*)
	PRM_Tim_Purge:				TIME;	(*durée du maintien pompage primaire en purge*)
	PRM_Tim_Arret_PP11:			TIME;	(*durée avant arrêt de la pompe primaire*)
	PRM_Tim_Int_BalInt:			TIME;	(*durée de pompage interjoint dans la phase d'alternance pompage interjoint/balayage pompe primaire*)
	PRM_Tim_Bal_BalInt:			TIME;	(*durée de balayage pompe primaire dans la phase d'alternance pompage interjoint/balayage pompe primaire*)
	PRM_Tim_FinBal:				TIME;	(*durée de balayage pompe primaire avant d'éteindre la pompe*)
	PRM_Pr_Atm:					REAL;	(*Pression atmosphérique dans l'enceinte*)
	PRM_Pr_PPrim:				REAL;	(*Pression de fin de pompage primaire dans l'enceinte*)
	PRM_Pr_RP_PPrim:			REAL;	(*Pression max admissible dans l'enceinte en pompage secondaire dans l'enceinte*)
	PRM_Pr_TGF:					REAL;	(*Pression de détection trés grosse fuite dans l'enceinte*)
	PRM_N_Purge:				USINT;	(*Nombre de cycles de purge pompage/ventilation*)
	CONF_Pompage_interjoint:	BOOL;	(*SPECIF 14035 non utilisé - Utilisation de la pompe primaire pour le pompage interjoint sur l'enceinte*)
	CONF_VINT:					BOOL;	(*SPECIF 14035 non utilisé - Utilisation d'une vanne d'isolement sur le pompage interjoint*)
	CONF_Volume_Enceinte:		REAL;	(*Volume pour RP*)

	PRM_Tim_Prep_Ventil:		TIME;	(*temporisation de prép ventilation (eau chaude suffisemment longtemps) *)

	(*Entité*)
	IsAssembly:		BOOL;		(*entité : ensemble*)
	IdXML:			STRING;		(*nom entité : identifiant pour recherche dans dico*)
	TagXML:			UINT;		(*nom entité : identifiant pour recherche dans dico*)
	IdParent:		STRING;		(*MNEMO de l'appelant*)
	MNEMO:			STRING;		(*MNEMO de l'entité*)
END_VAR


VAR_OUTPUT
	RQ_Prep_Ventil_Enc:		BOOL;											(*demande de préparation avant ventilation (réchauffement, arrêt eau ....*)
	RQ_Stop_Mesure_Enc:		BOOL;											(*demande d'arrêt de la mesure avant ventilation - Les blocs jauges concernés utilise		
																					cette information pour stoppée les jauges préalablement à la ventilation*)
END_VAR

VAR_IN_OUT
END_VAR

VAR
	VAR_Reset_Sortie:					BOOL;
	TIMER_SurVentilation_Enc:			TON;		(*Temporistion de surventilation enceinte*)
	TIMER_Purge:						TON;		(*Temporisation de maintien pompage primaire en purge*)
	TIMER_BalInt:						TON;		(*Temporisation gestion pompage interjoint et balayage pompe primaire*)
	TIMER_Arret_Roots:					TON;		(*Temporisation arrêt roots après prévidage*)
	TIMER_Arret_PP11:					TON;		(*Temporisation arrêt pompe primaire*)
	VAR_mem_isolement:					BOOL;
	VAR_Iter_Purge:						USINT;

	(*Pour RP*)
	VAR_Mem_Pression_Deb:		REAL;
	VAR_Mem_Pression_Fin:		REAL;
	VAR_Indicateur_Test:		REAL; 		(*résultat final*)
	TIMER_attente_test:			TON;		(*Temporisation pour test de remontée en pression*)
	FM_etape4:					R_TRIG;

	(*Pour prep ventil*)
	TIM_Prep_ventil:			TON;		(*timer de préparation ventil*)

	(*Pour regen*)
	FM_REGEN:					R_TRIG;		(* FM pompe cryogénique en régénération*)
	FD_REGEN:					F_TRIG;		(* FD pompe cryogénique en régénération*)
	TIMER_Post_Purge:			TON;		(*tempo max attente de retombée température après purge en regen partielle*)
	TIMER_etape6_regen:			TON;
	
	(*pour gestion pompage interjoint et vanne balayage pompe primaire*)
	VAR_BalInt:					BOOL;		(*conditions pour alternance interjoint/balayage : pompage secondaire sans puissance/chauffage/evap*)
	VAR_FinBal:					BOOL;		(*conditions pour balayage pompe primaire temporisé : avant d'arrêter la pompe*)
	VAR_Bal:					BOOL;		(*conditions pour balayage pompe primaire : pompe à l'arrêt*)
	VAR_Int:					BOOL;		(*conditions pour pompage interjoint : pas de regen, pompe en marche, pas de prévidage ou vide <100mbar*)
	VAR_BalInt_Ec:				BOOL;		
	VAR_Int_Ec:					BOOL;
	VAR_Int_Ok:					BOOL;
	VAR_FinBal_Ec:				BOOL;
	VAR_FinBal_Ok:				BOOL;
	VAR_Bal_Ec:					BOOL;
	VAR_No_Bal_Int_Ec:			BOOL;
END_VAR

PRL();

(*appel des opérations*)
ACT_ARRET_POMPES();
ACT_ISOLEMENT();
ACT_MARCHE_POMPES();
ACT_POMPAGE_PRIM();
ACT_POMPAGE_PROC();
ACT_POMPAGE_SEC();
ACT_VENTILATION();
ACT_PURGE();
ACT_REGEN();
ACT_REGEN_PART();
ACT_TEST_RP();
ACT_BAL_INT();

(*action en sortie*)
POST();

ACTION ACT_ARRET_POMPES:
(* OPERATION ARRET POMPES*)
(* arrêt des pompes*)

(*initialisation de l'opération*)
OP_ARRET_POMPES(
	CTRL_PLC:= CTRL_PLC,
	RESET:= RESET,
	ENABLE_INT:=TRUE,
	MANUAL:= MANUAL,
	ON_AUTO_INT:= (PP11.STATE_NOK AND PR11.STATE_NOK) AND (NOT OP_Pompage_Prim.Etape.0 OR NOT OP_Purge.Etape.0),
	RESTART_ENABLE_IF_OK:= FALSE,
	N_STEP_OP_OK:= 7,
	N_STEP_OP_NOK:=0);

(*appel de l'action de préparation de l'opération*)
OP_ARRET_POMPES.PRL();


(*GRAFCET*)
(* initialisation du grafcet*)
IF 		OP_Arret_Pompes.ETAPE = 0 THEN
				OP_Arret_Pompes.ETAPE.0 := TRUE;
(*repositionnement sur étape 0*)
ELSIF	MANUAL OR RESET OR OP_Marche_Pompes.ETAPE.1 THEN
				OP_Arret_Pompes.ETAPE := 0;			(*RAZ grafcet*)
				OP_Arret_Pompes.ETAPE.0:=TRUE;
(*étape 0-1*)
ELSIF 	OP_Arret_Pompes.ETAPE.0
		AND OP_Arret_Pompes.MARCHE_OP THEN
				OP_Arret_Pompes.ETAPE.1:=TRUE;
				OP_Arret_Pompes.ETAPE.0:=FALSE;
(*étape 1-2*)
ELSIF	OP_Arret_Pompes.ETAPE.1
		AND OP_Marche_Pompes.ETAPE.0  THEN
				OP_Arret_Pompes.Etape.2:=TRUE;
				OP_Arret_Pompes.Etape.1:=FALSE;
(*étape 2-3*)
ELSIF 	OP_Arret_Pompes.Etape.2
		AND (OP_Isolement.OK OR VAR_mem_isolement)
		AND (VINT.STATE_Off OR NOT CONF_VINT)
		 THEN
				OP_Arret_Pompes.Etape.3:=TRUE;
				OP_Arret_Pompes.Etape.2:=FALSE;
(*étape 3-4*)
ELSIF 	OP_Arret_Pompes.Etape.3
		AND	Timer_Arret_PP11.Q THEN 
				OP_Arret_Pompes.Etape.4:=TRUE;
				OP_Arret_Pompes.Etape.3:=FALSE;
(*étape 4-5*)
ELSIF	OP_Arret_Pompes.Etape.4
		AND PR11.STATE_Off AND PS11.STATE_Ar THEN
				OP_Arret_Pompes.Etape.5:=TRUE;
				OP_Arret_Pompes.Etape.4:=FALSE;
(*étape 5-6*)
ELSIF	OP_Arret_Pompes.Etape.5
		AND VAR_FinBal_Ok THEN
				OP_Arret_Pompes.Etape.6:=TRUE;
				OP_Arret_Pompes.Etape.5:=FALSE;
(*étape 6-7*)
ELSIF	OP_Arret_Pompes.Etape.6
		AND PP11.STATE_Off THEN
				OP_Arret_Pompes.Etape.7:=TRUE;
				OP_Arret_Pompes.Etape.6:=FALSE;
END_IF;

(*cloture du traitement de l'opération*)
OP_Arret_Pompes.POST();

(************************************************************************)
(*Gestion de la mémoire de la demande d'isolement de l'enceinte*)
(************************************************************************)
IF 		OP_Ventilation.Etape.9 THEN
	VAR_mem_isolement	:=	TRUE;
ELSIF	NOT OP_Pompage_Prim.AR OR NOT OP_Pompage_Sec.AR OR NOT OP_Pompage_Proc.AR OR NOT OP_Purge.AR THEN
	VAR_mem_isolement	:=	FALSE;
END_IF
(*IF OP_Arret_pompes.Etape.2 AND (NOT OP_Pompage_Prim.Etape.0  OR NOT OP_Pompage_Proc.Etape.0 OR NOT OP_Pompage_Sec.Etape.0) THEN
	VAR_mem_isolement_enceinte := TRUE;
END_IF;
IF OP_Arret_pompes.Etape.0 OR OP_Arret_Pompes.Etape.3 THEN
	VAR_mem_isolement_enceinte := FALSE;
END_IF;*)
END_ACTION

ACTION ACT_BAL_INT:
//Alternance balayage/pompage interjoint lorsque la cryo est opérationnelle, la pompe primaire également, qu'il n'y a pas de prévidage et pas de puissance extérieure
//Prioritaire sur VAR_Int
VAR_BalInt	:=	NOT PS11.STATE_Regen 
				AND PP11.STATE_On AND NOT OP_Arret_Pompes.Etape.5
				AND VP11.STATE_Off 
				AND I_Cond_Bal_PP11_Ext;
//Pompage interjoint uniquement lorsque la cryo est opérationnelle, la pompe primaire également et pas de préviage ou pression inférieure à 100mbar
VAR_Int		:=	NOT PS11.STATE_Regen
				AND PP11.STATE_On AND OP_Marche_Pompes.OK 
				AND (VP11.STATE_Off OR TH_Ouv_VINT);
//Balayage sur un temps donné (PRM_Tim_FinBal) lors de la demande d'arrêt de la pompage primaire en mode auto
VAR_FinBal	:=	OP_Arret_Pompes.Etape.5;
//Balayage permanent lorsque la pompe primaire est éteinte*)
VAR_Bal		:= 	PP11.STATE_Off;

(*GRAFCET*)
(* initialisation du grafcet*)
IF 		G7_Bal_Int.etape = 0
		THEN
				G7_Bal_Int.etape.0 := TRUE;
				
(*repositionnement sur étape 0*)
ELSIF	MANUAL OR RESET
		THEN
				G7_Bal_Int.etape := 0;			(*RAZ grafcet*)
				G7_Bal_Int.etape.0:=TRUE;
				
(*repositionnement sur étape 2*)
ELSIF	NOT G7_Bal_Int.etape.0 AND NOT G7_Bal_Int.etape.1
		AND VAR_BalInt AND NOT VAR_Bal AND NOT VAR_FinBal
		AND NOT VAR_Int_Ec
		AND NOT VAR_BalInt_Ec
		THEN
				G7_Bal_Int.etape := 0;			(*RAZ grafcet*)
				G7_Bal_Int.etape.2:=TRUE;
(*repositionnement sur étape 10*)
ELSIF	NOT G7_Bal_Int.etape.0 AND NOT G7_Bal_Int.etape.1
		AND NOT VAR_BalInt AND VAR_Int AND NOT VAR_Bal AND NOT VAR_FinBal
		AND NOT VAR_Int_Ec AND NOT VAR_Int_Ok
		THEN
				G7_Bal_Int.etape := 0;			(*RAZ grafcet*)
				G7_Bal_Int.etape.10:=TRUE;
(*repositionnement sur étape 14*)
ELSIF	NOT G7_Bal_Int.etape.0 AND NOT G7_Bal_Int.etape.1
		AND NOT VAR_BalInt AND NOT VAR_Int AND NOT VAR_Bal AND VAR_FinBal
		AND NOT VAR_FinBal_Ec AND NOT VAR_FinBal_Ok
		THEN
				G7_Bal_Int.etape := 0;			(*RAZ grafcet*)
				G7_Bal_Int.etape.14:=TRUE;
(*repositionnement sur étape 20*)
ELSIF	NOT G7_Bal_Int.etape.0 AND NOT G7_Bal_Int.etape.1
		AND NOT VAR_BalInt AND NOT VAR_Int AND NOT VAR_Bal AND NOT VAR_FinBal
		AND NOT VAR_No_Bal_Int_Ec
		THEN
				G7_Bal_Int.etape := 0;			(*RAZ grafcet*)
				G7_Bal_Int.etape.20:=TRUE;
(*repositionnement sur étape 23*)
ELSIF	NOT G7_Bal_Int.etape.0 AND NOT G7_Bal_Int.etape.1
		AND NOT VAR_BalInt AND NOT VAR_Int AND VAR_Bal AND NOT VAR_FinBal
		AND NOT VAR_Bal_Ec
		THEN
				G7_Bal_Int.etape := 0;			(*RAZ grafcet*)
				G7_Bal_Int.etape.23:=TRUE;
				
(*étape 0-1*)
ELSIF 	G7_Bal_Int.etape.0
		AND NOT MANUAL AND NOT RESET
		THEN
				G7_Bal_Int.etape.1:=TRUE;
				G7_Bal_Int.etape.0:=FALSE;
				
(*ALTERNANCE BALAYAGE / INTERJOINT*)
(*étape 1-2*)
ELSIF	G7_Bal_Int.etape.1
		AND VAR_BalInt AND NOT VAR_FinBal
		THEN
				G7_Bal_Int.etape.2:=TRUE;
				G7_Bal_Int.etape.1:=FALSE;
(*étape 2-3*)
ELSIF	G7_Bal_Int.etape.2
		AND VINT.STATE_Off
		THEN
				G7_Bal_Int.etape.3:=TRUE;
				G7_Bal_Int.etape.2:=FALSE;
(*étape 3-4*)
ELSIF	G7_Bal_Int.etape.3
		AND VN2PP11.STATE_On
		THEN
				G7_Bal_Int.etape.4:=TRUE;
				G7_Bal_Int.etape.3:=FALSE;
(*étape 3-4*)
ELSIF	G7_Bal_Int.etape.3
		AND VN2PP11.STATE_On
		THEN
				G7_Bal_Int.etape.4:=TRUE;
				G7_Bal_Int.etape.3:=FALSE;
(*étape 4-5*)
ELSIF	G7_Bal_Int.etape.4
		AND TIMER_BalInt.Q
		THEN
				G7_Bal_Int.etape.5:=TRUE;
				G7_Bal_Int.etape.4:=FALSE;
(*étape 5-6*)
ELSIF	G7_Bal_Int.etape.5
		AND VN2PP11.STATE_Off
		THEN
				G7_Bal_Int.etape.6:=TRUE;
				G7_Bal_Int.etape.5:=FALSE;
(*étape 6-7*)
ELSIF	G7_Bal_Int.etape.6
		AND VINT.STATE_On
		THEN
				G7_Bal_Int.etape.7:=TRUE;
				G7_Bal_Int.etape.6:=FALSE;
(*étape 7-2*)
ELSIF	G7_Bal_Int.etape.7
		AND TIMER_BalInt.Q
		THEN
				G7_Bal_Int.etape.2:=TRUE;
				G7_Bal_Int.etape.7:=FALSE;
				
				
(*INTERJOINT UNIQUEMENT*)
(*étape 1-10*)
ELSIF	G7_Bal_Int.etape.1
		AND NOT VAR_BalInt AND VAR_Int AND NOT VAR_Bal AND NOT VAR_FinBal
		THEN
				G7_Bal_Int.etape.10:=TRUE;
				G7_Bal_Int.etape.1:=FALSE;
(*étape 10-11*)
ELSIF	G7_Bal_Int.etape.10
		AND VN2PP11.STATE_Off
		THEN
				G7_Bal_Int.etape.11:=TRUE;
				G7_Bal_Int.etape.10:=FALSE;
(*étape 11-12*)
ELSIF	G7_Bal_Int.etape.11
		AND VINT.STATE_On
		THEN
				G7_Bal_Int.etape.12:=TRUE;
				G7_Bal_Int.etape.11:=FALSE;
							
				
(*BALAYAGE UNIQUEMENT - TEMPORISE*)
(*étape 1-14*)
ELSIF	G7_Bal_Int.etape.1
		AND NOT VAR_BalInt AND NOT VAR_Int AND NOT VAR_Bal AND VAR_FinBal
		THEN
				G7_Bal_Int.etape.14:=TRUE;
				G7_Bal_Int.etape.1:=FALSE;
(*étape 14-15*)
ELSIF	G7_Bal_Int.etape.14
		AND VINT.STATE_Off
		THEN
				G7_Bal_Int.etape.15:=TRUE;
				G7_Bal_Int.etape.14:=FALSE;
(*étape 15-16*)
ELSIF	G7_Bal_Int.etape.15
		AND VN2PP11.STATE_On
		THEN
				G7_Bal_Int.etape.16:=TRUE;
				G7_Bal_Int.etape.15:=FALSE;
(*étape 16-17*)
ELSIF	G7_Bal_Int.etape.16
		AND TIMER_BalInt.Q
		THEN
				G7_Bal_Int.etape.17:=TRUE;
				G7_Bal_Int.etape.16:=FALSE;
(*étape 17-18*)
ELSIF	G7_Bal_Int.etape.17
		AND VN2PP11.STATE_Off
		THEN
				G7_Bal_Int.etape.18:=TRUE;
				G7_Bal_Int.etape.17:=FALSE;
								
						
(*PAS DE BALAYAGE NI INTERJOINT*)
(*étape 1-20*)
ELSIF	G7_Bal_Int.etape.1
		AND NOT VAR_BalInt AND NOT VAR_Int AND NOT VAR_Bal AND NOT VAR_FinBal
		THEN
				G7_Bal_Int.etape.20:=TRUE;
				G7_Bal_Int.etape.1:=FALSE;
(*étape 20-21*)
ELSIF	G7_Bal_Int.etape.20
		AND VINT.STATE_Off AND VN2PP11.STATE_OFF
		THEN
				G7_Bal_Int.etape.21:=TRUE;
				G7_Bal_Int.etape.20:=FALSE;
				
				
(*BALAYAGE UNIQUEMENT - PERMANENT*)
(*étape 1-23*)
ELSIF	G7_Bal_Int.etape.1
		AND NOT VAR_BalInt AND NOT VAR_Int AND VAR_Bal AND NOT VAR_FinBal
		THEN
				G7_Bal_Int.etape.23:=TRUE;
				G7_Bal_Int.etape.1:=FALSE;
(*étape 23-24*)
ELSIF	G7_Bal_Int.etape.23
		AND VINT.STATE_Off
		THEN
				G7_Bal_Int.etape.24:=TRUE;
				G7_Bal_Int.etape.23:=FALSE;
(*étape 24-25*)
ELSIF	G7_Bal_Int.etape.24
		AND VN2PP11.STATE_On
		THEN
				G7_Bal_Int.etape.25:=TRUE;
				G7_Bal_Int.etape.24:=FALSE;
END_IF;

G7_Bal_Int.POST();

VAR_BalInt_Ec		:=	G7_Bal_Int.Etape.2 OR G7_Bal_Int.Etape.3 OR G7_Bal_Int.Etape.4 OR G7_Bal_Int.Etape.5 OR G7_Bal_Int.Etape.6 OR G7_Bal_Int.Etape.7;
VAR_Int_Ec			:=	G7_Bal_Int.Etape.10 OR G7_Bal_Int.Etape.11;
VAR_Int_Ok			:=	G7_Bal_Int.Etape.12;
VAR_FinBal_Ec		:=	G7_Bal_Int.Etape.14 OR G7_Bal_Int.Etape.15 OR G7_Bal_Int.Etape.16 OR G7_Bal_Int.Etape.17;
VAR_FinBal_Ok		:=	G7_Bal_Int.Etape.18;
VAR_No_Bal_Int_Ec	:=	G7_Bal_Int.Etape.20 OR G7_Bal_Int.Etape.21;
VAR_Bal_Ec			:=	G7_Bal_Int.Etape.23 OR G7_Bal_Int.Etape.24 OR G7_Bal_Int.Etape.25;
END_ACTION

ACTION ACT_ISOLEMENT:
(*OPERATION ISOLEMENT ENCEINTE*)
(*isolement de l'enceinte*)

(*initialisation de l'opération*)
OP_Isolement(
	CTRL_PLC:= CTRL_PLC,
	RESET:= RESET,
	ENABLE_INT:=TRUE,
	MANUAL:= MANUAL,
	ON_AUTO_INT:= 	((DEF_TGF.DEF OR DEF_RP_enc.DEF) AND (NOT OP_Pompage_Prim.Etape.0 OR NOT OP_Pompage_Sec.Etape.0 OR NOT OP_Pompage_proc.Etape.0))
					OR (PS11.STATE_Nok AND (NOT OP_Pompage_Sec.Etape.0 OR NOT OP_Pompage_proc.Etape.0))
					OR (PP11.STATE_Nok AND NOT OP_Pompage_Prim.Etape.0)
					OR (PR11.STATE_NOK AND NOT OP_Pompage_Prim.Etape.0),
	RESTART_ENABLE_IF_OK:= FALSE,
	N_STEP_OP_OK:= 4,
	N_STEP_OP_NOK:=0);

(*appel de l'action de préparation de l'opération*)
OP_Isolement.PRL();


(*GRAFCET*)
(* initialisation du grafcet*)
IF 		OP_Isolement.Etape = 0
		THEN
				OP_Isolement.Etape.0	:= TRUE;
(*repositionnement sur étape 0*)
ELSIF	MANUAL OR RESET OR OP_pompage_sec.Etape.1 OR OP_Pompage_Proc.Etape.1 OR Op_Pompage_Prim.Etape.1
		OR OP_ventilation.Etape.2 OR OP_Ventilation.Etape.9 OR OP_Purge.Etape.1 THEN
				OP_Isolement.Etape := 0;
				OP_Isolement.Etape.0:=TRUE;
(*étape 0-1*)
ELSIF 	OP_Isolement.Etape.0
		AND(
		OP_Isolement.Marche_OP OR
		OP_ventilation.Etape.1 OR
		OP_Test_RP.Etape.3 OR
		(OP_Arret_Pompes.Etape.2 AND NOT VAR_mem_isolement) OR
		OP_Regen.Etape.2 OR OP_Regen_Part.Etape.2
		)
		THEN
				OP_Isolement.Etape.1:=TRUE;
				OP_Isolement.Etape.0:=FALSE;
(*étape 1-2*)
ELSIF	OP_Isolement.Etape.1
		AND OP_Pompage_Proc.Etape.0
		AND OP_Pompage_Prim.Etape.0
		AND OP_Pompage_Sec.Etape.0
		AND (OP_Ventilation.Etape.0 OR OP_Ventilation.Etape.1)
		AND (OP_Purge.Etape.0 OR (OP_Purge.Etape.4 AND OP_Ventilation.Etape.1))
		THEN
				OP_Isolement.Etape.2:=TRUE;
				OP_Isolement.Etape.1:=FALSE;
(*étape 2-3*)
ELSIF 	OP_Isolement.Etape.2 AND
		VP11.STATE_Off AND
		VS11.STATE_Off AND
		VH11.STATE_Off  THEN
				OP_Isolement.Etape.3:=TRUE;
				OP_Isolement.Etape.2:=FALSE;
(*étape 3-4*)
ELSIF	OP_Isolement.Etape.3
		AND ((PP11.STATE_Off AND PR11.STATE_Off) OR PS11.STATE_Regen OR CONF_Pompage_interjoint) THEN
				OP_isolement.Etape.4:=TRUE;
				OP_isolement.Etape.3:=FALSE;
END_IF;

(*cloture du traitement de l'opération*)
OP_Isolement.POST();
END_ACTION

ACTION ACT_MARCHE_POMPES:
(* OPERATION MARCHE POMPES*)
(* mise en marche des pompes*)

(*initialisation de l'opération*)
OP_MARCHE_POMPES(
	CTRL_PLC:= CTRL_PLC,
	RESET:= RESET,
	ENABLE_INT:=TRUE,
	MANUAL:= MANUAL,
	ON_AUTO_INT:= TRUE,
	RESTART_ENABLE_IF_OK:= FALSE,
	N_STEP_OP_OK:= 5,
	N_STEP_OP_NOK:=0);

(*appel de l'action de préparation de l'opération*)
OP_MARCHE_POMPES.PRL();


(*GRAFCET*)
(* initialisation du grafcet*)
IF 		OP_MARCHE_POMPES.ETAPE = 0
		THEN
				OP_MARCHE_POMPES.ETAPE.0 := TRUE;
(*repositionnement sur étape 0*)
ELSIF	MANUAL OR RESET OR OP_ARRET_POMPES.ETAPE.1
		THEN
				OP_MARCHE_POMPES.ETAPE := 0;			(*RAZ grafcet*)
				OP_MARCHE_POMPES.ETAPE.0:=TRUE;
(*étape 0-1*)
ELSIF 	OP_MARCHE_POMPES.ETAPE.0
		AND (OP_MARCHE_POMPES.MARCHE_OP OR OP_POMPAGE_SEC.ETAPE.2
			OR (OP_Regen.Etape.5 AND TH_Atm))
		THEN
				OP_MARCHE_POMPES.ETAPE.1:=TRUE;
				OP_MARCHE_POMPES.ETAPE.0:=FALSE;
(*étape 1-2*)
ELSIF	OP_MARCHE_POMPES.ETAPE.1
		AND OP_ARRET_POMPES.ETAPE.0 AND PR11.STATE_Off AND I_Ref_Ok
		THEN
				OP_MARCHE_POMPES.ETAPE.2:=TRUE;
				OP_MARCHE_POMPES.ETAPE.1:=FALSE;
(*étape 2-3*)
ELSIF 	OP_MARCHE_POMPES.ETAPE.2
		AND (PP11.STATE_On OR NOT CONF_Pompage_interjoint)
		THEN
				OP_MARCHE_POMPES.ETAPE.3:=TRUE;
				OP_MARCHE_POMPES.ETAPE.2:=FALSE;
(*étape 3-4*)
ELSIF	OP_MARCHE_POMPES.ETAPE.3
		THEN
				OP_MARCHE_POMPES.ETAPE.4:=TRUE;
				OP_MARCHE_POMPES.ETAPE.3:=FALSE;
(*étape 4-5*)
ELSIF 	OP_MARCHE_POMPES.ETAPE.4
		AND PS11.STATE_On AND PS11.STATE_Ok AND NOT PS11.STATE_Regen
		THEN
				OP_MARCHE_POMPES.ETAPE.5:=TRUE;
				OP_MARCHE_POMPES.ETAPE.4:=FALSE;
(*étape 5-4*)
ELSIF 	OP_MARCHE_POMPES.ETAPE.5
		AND (PS11.STATE_Regen OR NOT PS11.STATE_Ok)		THEN
				OP_MARCHE_POMPES.ETAPE.4:=TRUE;
				OP_MARCHE_POMPES.ETAPE.5:=FALSE;
END_IF;

(*cloture du traitement de l'opération*)
OP_MARCHE_POMPES.POST();
END_ACTION

ACTION ACT_POMPAGE_PRIM:
(*OPERATION POMPAGE PRIMAIRE ENCEINTE*)
(*pompage primaire dans l'enceinte*)

(*initialisation de l'opération*)
OP_POMPAGE_PRIM(
	CTRL_PLC:= CTRL_PLC,
	RESET:= RESET,
	ENABLE_INT:= OP_Purge.Etape.0 AND IN_FE11T AND IN_FE12T,
	MANUAL:= MANUAL,
	RESTART_ENABLE_IF_OK:= FALSE,
	N_STEP_OP_OK:= 5,
	N_STEP_OP_NOK:=0);

(*appel de l'action de préparation de l'opération*)
OP_POMPAGE_PRIM.PRL();


(*GRAFCET*)
(* initialisation du grafcet*)
IF 		OP_Pompage_Prim.Etape = 0
		THEN
				OP_Pompage_Prim.Etape.0:= TRUE;
(*repositionnement sur étape 0*)
ELSIF	MANUAL OR RESET OR OP_Isolement.Etape.1 OR OP_Pompage_Sec.Etape.4
		OR OP_Pompage_Proc.Etape.1
		THEN
				OP_Pompage_Prim.ETAPE := 0;
				OP_Pompage_Prim.Etape.0:=TRUE;
(*étape 0-1*)
ELSIF 	OP_Pompage_Prim.Etape.0
		AND (OP_Pompage_Prim.Marche_OP OR OP_Pompage_Sec.Etape.3 OR OP_Purge.Etape.2)
		THEN
				OP_Pompage_Prim.Etape.1:=TRUE;
				OP_Pompage_Prim.Etape.0:=FALSE;
(*étape 1-2*)
ELSIF	OP_Pompage_Prim.Etape.1
		AND OP_Isolement.Etape.0
		AND OP_Ventilation.Etape.0
		AND OP_Pompage_Proc.Etape.0
		AND (OP_Pompage_Sec.Etape.0 OR OP_Pompage_Sec.Etape.3)
		AND (OP_Purge.Etape.0 OR OP_Purge.Etape.6 OR OP_Purge.Etape.2)
		AND VS11.STATE_Off
		AND VH11.STATE_Off
		THEN
				OP_Pompage_Prim.Etape.2:=TRUE;
				OP_Pompage_Prim.Etape.1:=FALSE;

(*étape 2-3*)
ELSIF 	OP_Pompage_prim.Etape.2
		THEN
				OP_Pompage_Prim.Etape.3:=TRUE;
				OP_Pompage_Prim.Etape.2:=FALSE;
(*étape 3-4*)
ELSIF	OP_Pompage_Prim.Etape.3
		AND PP11.STATE_On AND PR11.STATE_On THEN
				OP_Pompage_Prim.Etape.4:=TRUE;
				OP_Pompage_Prim.Etape.3:=FALSE;
(*étape 4-5*)
ELSIF 	OP_Pompage_Prim.Etape.4
		AND VP11.STATE_On
		THEN
				OP_Pompage_Prim.Etape.5:=TRUE;
				OP_Pompage_Prim.Etape.4:=FALSE;
END_IF;

(*cloture du traitement de l'opération*)
OP_Pompage_Prim.POST();
END_ACTION

ACTION ACT_POMPAGE_PROC:
(*OPERATION POMPAGE PROCEDE*)
(*pompage procede dans l'enceinte*)

(*initialisation de l'opération*)
OP_Pompage_Proc(
	CTRL_PLC:= CTRL_PLC,
	RESET:= RESET,
	ENABLE_INT:= OP_POMPAGE_SEC.OK OR OP_Pompage_Proc.OK,
	MANUAL:= MANUAL,
	RESTART_ENABLE_IF_OK:= FALSE,
	N_STEP_OP_OK:= 3,
	N_STEP_OP_NOK:=0);

(*appel de l'action de préparation de l'opération*)
OP_Pompage_Proc.PRL();


(*GRAFCET*)
(* initialisation du grafcet*)
IF 		OP_Pompage_Proc.Etape = 0
		THEN
				OP_Pompage_Proc.Etape.0:= TRUE;
(*repositionnement sur étape 0*)
ELSIF	MANUAL OR RESET OR OP_Isolement.Etape.1 OR OP_Pompage_Prim.Etape.1 OR OP_Pompage_Sec.Etape.1
		OR OP_Purge.Etape.1
		THEN
				OP_Pompage_Proc.Etape := 0;
				OP_Pompage_Proc.Etape.0:=TRUE;
(*étape 0-1*)
ELSIF 	OP_Pompage_Proc.Etape.0
		AND OP_Pompage_Proc.Marche_OP
		THEN
				OP_Pompage_Proc.Etape.1:=TRUE;
				OP_Pompage_Proc.Etape.0:=FALSE;
(*étape 1-2*)
ELSIF	OP_Pompage_Proc.Etape.1
		AND OP_Pompage_Sec.Etape.0
		THEN
				OP_Pompage_Proc.Etape.2:=TRUE;
				OP_Pompage_Proc.Etape.1:=FALSE;
(*étape 2-3*)
ELSIF 	OP_Pompage_proc.Etape.2
		AND VS11.STATE_Lam THEN
				OP_Pompage_Proc.Etape.3:=TRUE;
				OP_Pompage_Proc.Etape.2:=FALSE;
(*étape 3-2*)
ELSIF 	OP_Pompage_Proc.Etape.3
		AND OP_Pompage_Proc.Marche_OP
		THEN
				OP_Pompage_Proc.Etape.2:=TRUE;
				OP_Pompage_Proc.Etape.3:=FALSE;
END_IF;

(*cloture du traitement de l'opération*)
OP_Pompage_Proc.POST();
END_ACTION

ACTION ACT_POMPAGE_SEC:
(*OPERATION POMPAGE SECONDAIRE ENCEINTE*)
(*pompage secondaire dans l'enceinte*)

(*initialisation de l'opération*)
OP_pompage_sec(
	CTRL_PLC:= CTRL_PLC,
	RESET:= RESET,
	ENABLE_INT:=IN_FE11T AND IN_FE12T AND NOT PS11.STATE_Regen,
	MANUAL:= MANUAL,
	RESTART_ENABLE_IF_OK:= FALSE,
	N_STEP_OP_OK:= 7,
	N_STEP_OP_NOK:=0);

(*appel de l'action de préparation de l'opération*)
OP_Pompage_Sec.PRL();


(*GRAFCET*)
(* initialisation du grafcet*)
IF 		OP_Pompage_Sec.Etape = 0
		THEN
				OP_Pompage_Sec.Etape.0:= TRUE;
(*repositionnement sur étape 0*)
ELSIF	MANUAL OR RESET OR OP_Isolement.Etape.1 OR OP_Pompage_Proc.Etape.1
		OR (OP_Pompage_Prim.Etape.1 AND NOT OP_Pompage_Sec.Etape.3) OR OP_Purge.Etape.1
		THEN
				OP_Pompage_Sec.Etape := 0;
				OP_Pompage_Sec.Etape.0:=TRUE;
(*étape 0-1*)
ELSIF 	OP_Pompage_Sec.Etape.0 AND
		(OP_Pompage_Sec.Marche_OP OR OP_Purge.Etape.6 OR
			OP_Test_RP.Etape.2 OR OP_Test_RP.Etape.7
		OR (OP_Regen.Etape.5 AND NOT TH_Atm AND OP_Pompage_Sec.ENABLE_INT))
		THEN
				OP_Pompage_Sec.Etape.1:=TRUE;
				OP_Pompage_Sec.Etape.0:=FALSE;
(*étape 1-2*)
ELSIF	OP_Pompage_Sec.Etape.1
		AND OP_Isolement.Etape.0
		AND OP_Ventilation.Etape.0
		AND OP_Pompage_Proc.Etape.0
		AND (OP_Purge.Etape.0 OR OP_Purge.Etape.6)
		THEN
				OP_Pompage_Sec.Etape.2:=TRUE;
				OP_Pompage_Sec.Etape.1:=FALSE;
(*étape 2-3*)
ELSIF 	OP_Pompage_Sec.Etape.2
		AND OP_MARCHE_POMPES.ok AND NOT TH_Vide_Primaire AND VH11.STATE_Off
		THEN
				OP_Pompage_Sec.Etape.3:=TRUE;
				OP_Pompage_Sec.Etape.2:=FALSE;
(*étape 2-4*)
ELSIF 	OP_Pompage_Sec.Etape.2
		AND OP_MARCHE_POMPES.ok AND TH_Vide_Primaire AND VH11.STATE_Off
		THEN
				OP_Pompage_Sec.Etape.4:=TRUE;
				OP_Pompage_Sec.Etape.2:=FALSE;
(*étape 3-4*)
ELSIF	OP_Pompage_Sec.Etape.3
		AND	OP_POMPAGE_PRIM.ok  AND TH_Vide_Primaire
		THEN
				OP_Pompage_Sec.Etape.4:=TRUE;
				OP_Pompage_Sec.Etape.3:=FALSE;
(*étape 4-5*)
ELSIF	OP_Pompage_Sec.Etape.4
		AND VP11.STATE_Off
		AND  OP_POMPAGE_PRIM.AR   THEN
				OP_Pompage_Sec.Etape.5:=TRUE;
				OP_Pompage_Sec.Etape.4:=FALSE;
(*étape 5-6*)
ELSIF 	OP_Pompage_Sec.Etape.5
		AND (PP11.STATE_Off AND PR11.STATE_Off OR CONF_Pompage_interjoint)
		THEN
				OP_Pompage_Sec.Etape.6:=TRUE;
				OP_Pompage_Sec.Etape.5:=FALSE;
(*étape 6-7*)
ELSIF 	OP_Pompage_Sec.Etape.6
		AND VS11.STATE_On
		THEN
				OP_Pompage_Sec.Etape.7:=TRUE;
				OP_Pompage_Sec.Etape.6:=FALSE;
END_IF;

(*cloture du traitement de l'opération*)
OP_Pompage_Sec.POST();
END_ACTION

ACTION ACT_PURGE:
(*OPERATION PURGE*)
(*purge enceinte : pompage primaire pendant un temps donné puis ventilation, répété X fois*)

